// TwinCAT 3 PLC project PLC
// ProgramVersion: 3.1.4026.14
// CompilerDefines: VISU_USEPROPERTYINFO
// libraries:
//   Tc2_Standard, * (Beckhoff Automation GmbH)
//   Tc2_System, * (Beckhoff Automation GmbH)
//   Tc3_Analytics, * (Beckhoff Automation GmbH)
//   TcoCore, * (Vortex.Library)
//   TcoDrivesBeckhoff, * (Vortex.Library)
//   TcoElements, * (Vortex.Library)
//   TcoIo, * (Vortex.Library)
//   TcoPneumatics, * (Vortex.Library)
//   TcoUtilities, * (Vortex.Library)
//   VisuDialogs, * (System)
// project tree:
//   Components/ ST_MachineSetting.TcDUT (not stored)
//   Components/TcaCarrier/Structures/ TcaCarrierService.TcDUT (not stored), TcaCarrierConfig.TcDUT (not stored), TcaCarrierStatus.TcDUT
//   Components/TcaCarrier/Enumerations/ eTcaCarrierCmd.TcDUT (not stored), eTcaCarrierConfig.TcDUT (not stored)
//   Components/TcaCarrier/ ITcaCarrier.TcIO (not stored), TcaCarrier.TcPOU
//   Components/TcaCarrier/Tasks/ TcaCarrierModifyTask.TcPOU
//   Components/TcaPushButton/Enumerations/ eTcaPushButtonColor.TcDUT (not stored), eTcaPushButtonLightState.TcDUT (not stored)
//   Components/TcaPushButton/Structures/ TcaPushButtonStatus.TcDUT, TcaPushButtonRef.TcDUT, TcaPushButtonConfig.TcDUT, TcaPushButtonService.TcDUT (not stored)
//   Components/TcaPushButton/ TcaPushButton.TcPOU (not stored)
//   Components/TcaStorage/ E_ApproachDirection.TcDUT, eTcaStorageCmd.TcDUT (not stored), TcaRobotStorage.TcPOU (excluded from build), TcaStorage.TcPOU (not stored), TcaStorageRef.TcDUT (not stored)
//   Components/TcaTrolley/ CMD_Trolley.TcDUT (not stored), eTcaTrolleyCmd.TcDUT (not stored), TcaTrolley.TcPOU, TcaTrolleyRef.TcDUT
//   Components/TcaWorkpiecePlace/Enumerations/ eTcaWorkpiecePlaceProgress.TcDUT, eTcaWorkpiecePlaceStatus.TcDUT
//   Components/TcaWorkpiecePlace/Structures/ TcaWorkpiecePlaceService.TcDUT (not stored), TcaWorkpiecePlaceConfig.TcDUT, TcaWorkpiecePlaceStatus.TcDUT
//   Components/TcaWorkpiecePlace/ TcaWorkpiecePlace.TcPOU (not stored)
//   Components_RMTH/TcaEngelCasting/ Schnittstellenprotokoll.TcDUT (not stored), TcaEngelCastingCarrierInput.TcDUT (not stored), TcaEngelCastingCarrierJob.TcDUT (not stored), TcaEngelCastingCarrierJobStatus.TcDUT (not stored), TcaEngelCastingCarrierOutput.TcDUT (not stored), TcalEngelCastingCarrierStatus.TcDUT (not stored)
//   Components_RMTH/TcaLaserDistanceSenor/Structures/ TcaLaserDistanceSenorConfig.TcDUT, TcaLaserDistanceSenorRef.TcDUT (not stored), TcaLaserDistanceSenorStatus.TcDUT, TcaLaserDistanceSensorDataArrayEntry.TcDUT (not stored), TcaLaserDistanceSenorService.TcDUT
//   Components_RMTH/TcaLaserDistanceSenor/ TcaLaserDistanceSenor.TcPOU
//   Components_RMTH/TcaRackFeeder/Structures/ TcaRackFeederConfig.TcDUT, TcaRackFeederRef.TcDUT, TcaRackFeederService.TcDUT (not stored), TcaRackFeederStatus.TcDUT (not stored)
//   Components_RMTH/TcaRackFeeder/ TcaRackFeeder.TcPOU
//   Components_RMTH/TcaSafetyGate/ ISafetyComponent.TcIO (not stored), TcaSafetyGate.TcPOU (not stored)
//   Components_RMTH/TcaSafetyGate/Structures/ TcaSafetyGateConfig.TcDUT, TcaSafetyGateRef.TcDUT (not stored), TcaSafetyGateService.TcDUT (not stored), TcaSafetyGateStatus.TcDUT (not stored)
//   Components_RMTH/TcaSegmentDoor/Structures/ TcaSegmentDoorConfig.TcDUT, TcaSegmentDoorRef.TcDUT (not stored), TcaSegmentDoorService.TcDUT (not stored), TcaSegmentDoorStatus.TcDUT
//   Components_RMTH/TcaSegmentDoor/ TcaSegmentDoor.TcPOU (not stored)
//   Components_RMTH/TcaTwinSAFE/Structures/ TcaTwinSAFEConfig.TcDUT (not stored), TcaTwinSAFERef.TcDUT (not stored), TcaTwinSAFEService.TcDUT (not stored), TcaTwinSAFEStatus.TcDUT (not stored)
//   Components_RMTH/TcaTwinSAFE/ TcaTwinSAFE.TcPOU
//   / GlobalTextList.TcGTLO (not stored), PlcTask.TcTTO (not stored), Visualization Manager.TcVMO (not stored)
//   Items/ COLOR.TcDUT (not stored), E_Coordinate.TcDUT, ST_ComboboxEntry.TcDUT (not stored), ST_Coordinate.TcDUT, ST_WorkpieceType.TcDUT (not stored)
//   Program/Handling/Dialogs/ Handling_TeachRack_DlgContent.TcPOU (not stored)
//   Program/Handling/Sequences/ Handling_Teach.TcPOU, Handling_TeachRack.TcPOU, Handling_GroundMode.TcPOU (not stored), Handling_OpenDoor.TcPOU (not stored)
//   Program/ MAIN.TcPOU, Peripherie.TcPOU (not stored)
//   Program/Handling/ Handling.TcPOU (not stored), Handling_Components.TcPOU, Handling_Positions.TcPOU (not stored)
//   Template/Component_Cylinder/Base/ CylinderBase.TcPOU (not stored), TcoCylinderBase.TcPOU, TcoDoubleCylinderBase.TcPOU (not stored)
//   Template/Component_Cylinder/ ITcoCylinder.TcIO, TcoCylinder.TcPOU (not stored), TcoDoubleCylinder.TcPOU (not stored)
//   Template/Component_Cylinder/Structs/ CylinderConfig.TcDUT (not stored), CylinderStatus.TcDUT, TcoCylinderConfig.TcDUT (not stored), TcoCylinderStatus.TcDUT (not stored)
//   Template/Component_Cylinder/Tasks/ CylinderMoveTask.TcPOU (not stored), TcoCylinderMoveTask.TcPOU
//   Template/RackFeeder/ CMD_RackFeeder.TcDUT (not stored), E_RackFeederCmd.TcDUT, FB_RackFeeder.TcPOU (not stored)
//   Template/RackFeeder/Structure/ ST_RackFeederIO.TcDUT (not stored), ST_RackFeederJob.TcDUT (not stored), ST_StorageDock.TcDUT, ST_TrolleyDock.TcDUT
//   Template/Station/Data/ ST001_ProcessData.TcDUT, ST001_ProcessDataManager.TcPOU
//   Template/Station/ ST001.TcPOU (not stored), ST001_AutomatSequence.TcPOU, ST001_Components.TcDUT, ST001_ComponentsHandler.TcPOU (not stored), ST001_GroundSequence.TcPOU (not stored)
//   Template/Component_Carousell/Base/ TcoCarouselBase.TcPOU
//   Template/Component_Carousell/Structs/ eTcoCarouselDirection.TcDUT (not stored), TcoCarouselConfig.TcDUT (not stored), TcoCarouselStatus.TcDUT (not stored)
//   Template/Component_Carousell/Tasks/ TcoTurnTableTask.TcPOU (not stored)
//   Template/Component_Carousell/ TcoCarousel.TcPOU
//   Utilities/Component/Enumerations/ E_ComponentState.TcDUT (not stored), E_SafeState.TcDUT
//   Utilities/Component/ FB_Component.TcPOU (not stored), FB_ComponentPool.TcPOU
//   Utilities/Component/Interfaces/ ITF_Component.TcIO
//   Utilities/Component/Structures/ ST_ComponentVisu.TcDUT (not stored)
//   Utilities/Component/Visualisation/ Uc_Component.TcVIS
//   Utilities/EventLog/Base/ FB_LoggingProviderBase.TcPOU
//   Utilities/EventLog/Enumerations/ E_BoolFilter.TcDUT, E_FilterActive.TcDUT, E_LoggingProvider.TcDUT (not stored), E_LogLevel.TcDUT, E_Priority.TcDUT (not stored), ST_LoggingConfig.TcDUT
//   Utilities/EventLog/ E_Event.TcDUT (not stored), FB_EventLog.TcPOU (not stored)
//   Utilities/EventLog/Interface/ ITFLoggingProvider.TcIO (not stored), ITF_EventLog.TcIO
//   Utilities/EventLog/Structures/ ST_Event.TcDUT, ST_EventBase.TcDUT (not stored), ST_EventOutput.TcDUT, ST_EventVisu.TcDUT (not stored), ST_Log.TcDUT
//   Utilities/EventLog/Visualization/ Uc_EventLog.TcVIS, Uc_EventLogControl.TcDUT, Uc_EventLogControl.TcVIS, Uc_EventLogEntry.TcVIS, Uc_EventLogTable.TcDUT, Uc_EventLogTable.TcVIS
//   Utilities/Helpers/Color/ F_DWORD2CMYK.TcPOU, F_DWORD2RGB.TcPOU (not stored), F_RGB2CMYK.TcPOU (not stored), F_RGB2DWORD.TcPOU, F_TextColor.TcPOU (not stored), ST_Color.TcDUT, ST_ColorCMYK.TcDUT (not stored)
//   Utilities/Helpers/Concat/ Concat10.TcPOU, Concat2.TcPOU (not stored), Concat3.TcPOU, Concat4.TcPOU, Concat5.TcPOU, Concat6.TcPOU, Concat7.TcPOU (not stored), Concat8.TcPOU, Concat9.TcPOU, ConcatArray.TcPOU
//   Utilities/Helpers/ E_OperationResult.TcDUT (not stored), FB_GetTimeString.TcPOU (excluded from build), FB_Pulse.TcPOU, FB_TON_RMTH.TcPOU, F_BYTE_TO_INT.TcPOU, F_BYTE_TO_REAL.TcPOU (not stored), F_DT_TO_STRING.TcPOU (not stored), F_GetAdsPort.TcPOU (not stored), F_GetPlcCycleTime.TcPOU, F_GetSystemTime64.TcPOU, F_TO_STRING.TcPOU, P_FilePath.TcPOU (not stored), P_System.TcPOU, ST_DefaultPulse.TcDUT (not stored), ST_PlcSystemInfo.TcDUT (not stored)
//   Utilities/ HexColor.TcGVL, Statics.TcGVL, StaticsConstant.TcGVL (not stored)
//   Utilities/List/ FB_List.TcPOU (not stored)
//   Utilities/List/Structures/ ST_Listentry.TcDUT (not stored), Uc_List.TcDUT
//   Utilities/List/Visu/ Uc_EntryDetail.TcVIS (not stored), Uc_List.TcVIS, Uc_Listentry.TcVIS
//   Utilities/Sequencer/Enumeration/ E_SequenceState.TcDUT
//   Utilities/Sequencer/ FB_Sequence.TcPOU
// real-time tasks:
//   TASK PlcTask: cycle T#10ms, priority 20, ADS port 350
// motion (NC):
//   TASK NC-Task 1 SAF: cycle T#2ms, priority 4, ADS port 501
//   TASK NC-Task 1 SVB: cycle T#10ms, priority 8, ADS port 511
//   AXIS Oven B CH1 (id 14)
//     Dynamic: Acceleration=282800000, Deceleration=282800000, Jerk=2.85628e+17
//     Velo: RefSearch=25, RefSync=25, SlowManual=14, FastManual=28, Maximum=28
//     PositionAreaControl: Enable=false
//     TargetPosControl: Enable=false
//     OtherSettings: AllowMotionCmdToSlave=true
//     encoder EncType=7
//       EncPara: ScaleFactorNumerator=0.001879, Offset=-1.4, MaxCount=#x0000ffff, ReferenceSystem=1
//     drive DrvType=23
//       Analog: VeloReferenz=28, TorqueSetpointScale=10, ScaleFactorActTorque=0.1
//       TimeComp: TaskDelayCycles=1
//     controller CtrType=1
//       CtrPara: PriorControlFactor=1
//         PosDiffControl: Enable=false
//         Observer: BandWidth=20
//   AXIS Oven B CH2 (id 15)
//     Dynamic: Acceleration=282800000, Deceleration=282800000, Jerk=2.85628e+17
//     Velo: RefSearch=25, RefSync=25, SlowManual=14, FastManual=28, Maximum=28
//     PositionAreaControl: Enable=false
//     TargetPosControl: Enable=false
//     OtherSettings: AllowMotionCmdToSlave=true
//     encoder EncType=7
//       EncPara: ScaleFactorNumerator=0.001879, Offset=-1.4, MaxCount=#x0000ffff, ReferenceSystem=1
//     drive DrvType=23
//       Analog: VeloReferenz=28, TorqueSetpointScale=10, ScaleFactorActTorque=0.1
//       TimeComp: TaskDelayCycles=1
//     controller CtrType=1
//       CtrPara: PriorControlFactor=1
//         PosDiffControl: Enable=false
//         Observer: BandWidth=20
//   AXIS Rackfeeder X (id 16)
//     Dynamic: Acceleration=2461.9275, Deceleration=2461.9275, Jerk=7385.7825
//     Velo: RefSearch=16.41285, RefSync=16.41285, SlowManual=10, FastManual=60, Fast=1641.285, Maximum=1641.285
//     OtherSettings: AllowMotionCmdToSlave=true
//     encoder EncType=8
//       EncPara: ScaleFactorNumerator=150, ScaleFactorDenominator=10485760, MaxCount=#xffffffff
//     drive DrvType=9
//       DrvPara: MaxCount=#xffffffff, DriveControlDWord=#x00030100
//         Analog: VeloReferenz=1805.4135, VeloScale=1.02400649589962, TorqueSetpointScale=10, ScaleFactorActTorque=0.1
//         TimeComp: TaskDelayCycles=1
//     controller CtrType=1
//       CtrPara: PriorControlFactor=1
//         Observer: BandWidth=20
//   AXIS Rackfeeder Y (id 17)
//     Dynamic: Acceleration=2256.7665, Deceleration=2256.7665, Jerk=6770.2995
//     Velo: RefSearch=15.04511, RefSync=15.04511, SlowManual=10, FastManual=60, Fast=1504.511, Maximum=1504.511
//     OtherSettings: AllowMotionCmdToSlave=true
//     encoder EncType=8
//       EncPara: ScaleFactorNumerator=220, ScaleFactorDenominator=16777216, MaxCount=#xffffffff
//     drive DrvType=9
//       DrvPara: MaxCount=#xffffffff, DriveControlDWord=#x00030100
//         Analog: VeloReferenz=1654.9621, VeloScale=1.02400649589962, TorqueSetpointScale=10, ScaleFactorActTorque=0.1
//         TimeComp: TaskDelayCycles=1
//     controller CtrType=1
//       CtrPara: PriorControlFactor=1
//         Observer: BandWidth=20
//   AXIS Rackfeeder Teleskop (id 18)
//     OtherSettings: AllowMotionCmdToSlave=true
//     encoder EncType=8
//       EncPara: MaxCount=#xffffffff
//     drive DrvType=9
//       DrvPara: MaxCount=#xffffffff, DriveControlDWord=#x00030100
//         Analog: VeloScale=1.02400649589962, TorqueSetpointScale=10, ScaleFactorActTorque=0.1
//         TimeComp: TaskDelayCycles=1
//     controller CtrType=1
//       CtrPara: PriorControlFactor=1
//         Observer: BandWidth=20
//   AXIS Oven B (id 21)
//     Dynamic: Acceleration=1231.0125, Deceleration=1231.0125, Jerk=3693.0375
//     Velo: RefSearch=8.20675, RefSync=8.20675, SlowManual=20, FastManual=120, Fast=820.675, Maximum=820.675
//     OtherSettings: AllowMotionCmdToSlave=true
//     encoder EncType=8
//       EncPara: ScaleFactorNumerator=120, ScaleFactorDenominator=16777216, Inverse=true, MaxCount=#xffffffff
//     drive DrvType=9
//       DrvPara: Inverse=true, MaxCount=#xffffffff, DriveControlDWord=#x00030100
//         Analog: VeloReferenz=902.7425, VeloScale=1.02400649589962, TorqueSetpointScale=10, ScaleFactorActTorque=0.1
//         TimeComp: TaskDelayCycles=1
//     controller CtrType=1
//       CtrPara: PriorControlFactor=1
//         Observer: BandWidth=20
//   AXIS Oven A (id 20)
//     Dynamic: Acceleration=1231.0125, Deceleration=1231.0125, Jerk=3693.0375
//     Velo: RefSearch=8.20675, RefSync=8.20675, SlowManual=20, FastManual=120, Fast=820.675, Maximum=820.675
//     OtherSettings: AllowMotionCmdToSlave=true
//     encoder EncType=8
//       EncPara: ScaleFactorNumerator=120, ScaleFactorDenominator=16777216, Inverse=true, MaxCount=#xffffffff
//     drive DrvType=9
//       DrvPara: Inverse=true, MaxCount=#xffffffff, DriveControlDWord=#x00030100
//         Analog: VeloReferenz=902.7425, VeloScale=1.02400649589962, TorqueSetpointScale=10, ScaleFactorActTorque=0.1
//         TimeComp: TaskDelayCycles=1
//     controller CtrType=1
//       CtrPara: PriorControlFactor=1
//         Observer: BandWidth=20
//   AXIS Oven A CH1 (id 1)
//     Dynamic: Acceleration=282800000, Deceleration=282800000, Jerk=2.85628e+17, DelayTime=0.01, OverrideType=4
//     Velo: RefSearch=25, RefSync=25, SlowManual=14, FastManual=28, Maximum=28
//     PositionAreaControl: Enable=false
//     TargetPosControl: Enable=false
//     OtherSettings: AllowMotionCmdToSlave=true
//     encoder EncType=7
//       EncPara: ScaleFactorNumerator=0.001879, Offset=-1.4, EncMode=1, MaxCount=#x0000ffff, ReferenceSystem=1
//         FilterTime: TVelo=0.1
//         SoftEndMinControl: Range=-5
//         SoftEndMaxControl: Range=30
//         ActPosCorrection: Enable=true, Time=1
//     drive DrvType=23
//       Analog: VeloReferenz=28, TorqueSetpointScale=10, ScaleFactorActTorque=0.1
//       TimeComp: TaskDelayCycles=1
//     controller CtrType=1
//       CtrPara: PriorControlFactor=1
//         PosDiffControl: Enable=false
//         Observer: BandWidth=20
//   AXIS Oven A CH2 (id 13)
//     Dynamic: Acceleration=282800000, Deceleration=282800000, Jerk=2.85628e+17
//     Velo: RefSearch=25, RefSync=25, SlowManual=14, FastManual=28, Maximum=28
//     PositionAreaControl: Enable=false
//     TargetPosControl: Enable=false
//     OtherSettings: AllowMotionCmdToSlave=true
//     encoder EncType=7
//       EncPara: ScaleFactorNumerator=0.001879, Offset=-1.4, MaxCount=#x0000ffff, ReferenceSystem=1
//     drive DrvType=23
//       Analog: VeloReferenz=28, TorqueSetpointScale=10, ScaleFactorActTorque=0.1
//       TimeComp: TaskDelayCycles=1
//     controller CtrType=1
//       CtrPara: PriorControlFactor=1
//         PosDiffControl: Enable=false
//         Observer: BandWidth=20
// I/O:
//   DEVICE Gerät 3 (EtherCAT), AmsNetId 5.24.124.74.4.1
//     Klemme 1 (EK1100) [EK1100 EtherCAT-Koppler (2A E-Bus)]
//       Klemme 33 (EL6910) [EL6910, TwinSAFE PLC]
//       Klemme 3 (EL1904) [EL1904, 4 K. Safety Eingang 24V, TwinSAFE]
//         modules: Module 1 (FSOES)
//       Klemme 4 (EL2904) [EL2904, 4 K. Safety Ausgang 24V, 0.5A, TwinSAFE]
//         modules: Module 1 (FSOES), Module 2 (DO)
//       Klemme 5 (EL1104) [EL1104 4K. Dig. Eingang 24V, 3ms, Sensorversorgung]
//       Klemme 6 (EL1104) [EL1104 4K. Dig. Eingang 24V, 3ms, Sensorversorgung]
//       Klemme 7 (EL6224) [EL6224 (IO Link Master)]
//       ENGEL Interface (EL1008) [EL1008 8K. Dig. Eingang 24V, 3ms]
//       ENGEL Interface (EL2624) [EL2624 4K. Relais Ausgang, Schließer (125V AC / 30V DC)]
//       Ovens (EK1122) [EK1122 2-Port EtherCAT-Abzweig]
//         Oven_A (EK1100) [EK1100 EtherCAT-Koppler (2A E-Bus)]
//           Klemme 10 (EL1904) [EL1904, 4 K. Safety Eingang 24V, TwinSAFE]
//             modules: Module 1 (FSOES)
//           Klemme 11 (EL2904) [EL2904, 4 K. Safety Ausgang 24V, 0.5A, TwinSAFE]
//             modules: Module 1 (FSOES), Module 2 (DO)
//           Klemme 12 (EL7332) [EL7332 2K. DC-Motor-Endstufe (24V, 1.5A)]
//           Klemme 13 (EL3062-0030) [EL3062-0030 2K.Ana. Eingang 0-30V]
//           Klemme 14 (EL1004) [EL1004 4K. Dig. Eingang 24V, 3ms]
//           Klemme 15 (EL2004) [EL2004 4K. Dig. Ausgang 24V, 0.5A]
//           Klemme 16 (EL9010) [EL9010 Endklemme]
//         Oven_B (EK1100) [EK1100 EtherCAT-Koppler (2A E-Bus)]
//           Klemme 18 (EL1904) [EL1904, 4 K. Safety Eingang 24V, TwinSAFE]
//             modules: Module 1 (FSOES)
//           Klemme 19 (EL2904) [EL2904, 4 K. Safety Ausgang 24V, 0.5A, TwinSAFE]
//             modules: Module 1 (FSOES), Module 2 (DO)
//           Klemme 20 (EL7332) [EL7332 2K. DC-Motor-Endstufe (24V, 1.5A)]
//           Klemme 21 (EL3062-0030) [EL3062-0030 2K.Ana. Eingang 0-30V]
//           Klemme 22 (EL1004) [EL1004 4K. Dig. Eingang 24V, 3ms]
//           Klemme 23 (EL2004) [EL2004 4K. Dig. Ausgang 24V, 0.5A]
//           Klemme 61 (EL9010) [EL9010 Endklemme]
//       Storage|Casting (EK1122) [EK1122 2-Port EtherCAT-Abzweig]
//         Storage (EK1100)
//     RackFeeder_X_Y (AX5206-0000-0215) [AX5206-0000-0215 EtherCAT Drive (SoE, 2 Ch.)]
//       Klemme 27 (AX5805) [AX5805 (Safety Drive Option)]
//         modules: Module 1 (Safety Process Data, 2 axis), Module 2 (Standard Process Data, 2 axis)
//     Rackfeeder_Teleskop (AX5203-0000-0215) [AX5203-0000-0215 EtherCAT Drive (SoE, 2 Ch.)]
//       Klemme 29 (AX5805) [AX5805 (Safety Drive Option)]
//         modules: Module 1 (Safety Process Data, 2 axis), Module 2 (Standard Process Data, 2 axis)
//     OvenDoor_A_B (AX5206-0000-0215) [AX5206-0000-0215 EtherCAT Drive (SoE, 2 Ch.)]
//       Klemme 31 (AX5805) [AX5805 (Safety Drive Option)]
//         modules: Module 1 (Safety Process Data, 2 axis), Module 2 (Standard Process Data, 2 axis)
// variable links:
//   Device 3 (EtherCAT) <-> Device 3 (EtherCAT)/OvenDoor_A_B (AX5206-0000-0215)/Term 31 (AX5805)
//     Term 1 (EK1100)/Term 33 (EL6910)/ConnectionInputs/TwinSafeMain.Oven (AX5805) - Module 1 (Safety Process Data, 2 axis)_120 TxPDO <-> Module 1 (Safety Process Data, 2 axis)/Outputs (Controlword)/FSOE
//     Term 1 (EK1100)/Term 33 (EL6910)/ConnectionOutputs/TwinSafeMain.Oven (AX5805) - Module 1 (Safety Process Data, 2 axis)_120 RxPDO <-> Module 1 (Safety Process Data, 2 axis)/Inputs (Statusword)/FSOE
//   Device 3 (EtherCAT) <-> Device 3 (EtherCAT)/RackFeeder_X_Y (AX5206-0000-0215)/Term 27 (AX5805)
//     Term 1 (EK1100)/Term 33 (EL6910)/ConnectionInputs/TwinSafeMain.Rackfeeder_XY (AX5805) - Module 1 (Safety Process Data, 2 axis)_118 TxPDO <-> Module 1 (Safety Process Data, 2 axis)/Outputs (Controlword)/FSOE
//     Term 1 (EK1100)/Term 33 (EL6910)/ConnectionOutputs/TwinSafeMain.Rackfeeder_XY (AX5805) - Module 1 (Safety Process Data, 2 axis)_118 RxPDO <-> Module 1 (Safety Process Data, 2 axis)/Inputs (Statusword)/FSOE
//   Device 3 (EtherCAT) <-> Device 3 (EtherCAT)/Rackfeeder_Teleskop (AX5203-0000-0215)/Term 29 (AX5805)
//     Term 1 (EK1100)/Term 33 (EL6910)/ConnectionInputs/TwinSafeMain.Rackfeeder_Tele (AX5805) - Module 1 (Safety Process Data, 2 axis)_119 TxPDO <-> Module 1 (Safety Process Data, 2 axis)/Outputs (Controlword)/FSOE
//     Term 1 (EK1100)/Term 33 (EL6910)/ConnectionOutputs/TwinSafeMain.Rackfeeder_Tele (AX5805) - Module 1 (Safety Process Data, 2 axis)_119 RxPDO <-> Module 1 (Safety Process Data, 2 axis)/Inputs (Statusword)/FSOE
//   Device 3 (EtherCAT) <-> Device 3 (EtherCAT)/Term 1 (EK1100)/Ovens (EK1122)/Oven_A (EK1100)/Term 10 (EL1904)
//     Term 1 (EK1100)/Term 33 (EL6910)/ConnectionInputs/TwinSafeMain.Oven A (EL1904) - Module 1 (FSOES)_14 TxPDO <-> Module 1 (FSOES)/RxPDO/FSOE
//     Term 1 (EK1100)/Term 33 (EL6910)/ConnectionOutputs/TwinSafeMain.Oven A (EL1904) - Module 1 (FSOES)_14 RxPDO <-> Module 1 (FSOES)/TxPDO/FSOE
//   Device 3 (EtherCAT) <-> Device 3 (EtherCAT)/Term 1 (EK1100)/Ovens (EK1122)/Oven_A (EK1100)/Term 11 (EL2904)
//     Term 1 (EK1100)/Term 33 (EL6910)/ConnectionInputs/TwinSafeMain.Oven A (EL2904) - Module 1 (FSOES)_111 TxPDO <-> Module 1 (FSOES)/RxPDO/FSOE
//     Term 1 (EK1100)/Term 33 (EL6910)/ConnectionOutputs/TwinSafeMain.Oven A (EL2904) - Module 1 (FSOES)_111 RxPDO <-> Module 1 (FSOES)/TxPDO/FSOE
//   Device 3 (EtherCAT) <-> Device 3 (EtherCAT)/Term 1 (EK1100)/Ovens (EK1122)/Oven_B (EK1100)/Term 18 (EL1904)
//     Term 1 (EK1100)/Term 33 (EL6910)/ConnectionOutputs/TwinSafeMain.Oven B (EL1904) - Module 1 (FSOES)_16 RxPDO <-> Module 1 (FSOES)/TxPDO/FSOE
//   Device 3 (EtherCAT) <-> Device 3 (EtherCAT)/Term 1 (EK1100)/Ovens (EK1122)/Oven_B (EK1100)/Term 19 (EL2904)
//     Term 1 (EK1100)/Term 33 (EL6910)/ConnectionInputs/TwinSafeMain.Oven B (EL2904) - Module 1 (FSOES)_112 TxPDO <-> Module 1 (FSOES)/RxPDO/FSOE
//     Term 1 (EK1100)/Term 33 (EL6910)/ConnectionOutputs/TwinSafeMain.Oven B (EL2904) - Module 1 (FSOES)_112 RxPDO <-> Module 1 (FSOES)/TxPDO/FSOE
//   Device 3 (EtherCAT) <-> Device 3 (EtherCAT)/Term 1 (EK1100)/Term 3 (EL1904)
//     Term 1 (EK1100)/Term 33 (EL6910)/ConnectionInputs/TwinSafeMain.MAIN (EL1904) - Module 1 (FSOES)_12 TxPDO <-> Module 1 (FSOES)/RxPDO/FSOE
//     Term 1 (EK1100)/Term 33 (EL6910)/ConnectionOutputs/TwinSafeMain.MAIN (EL1904) - Module 1 (FSOES)_12 RxPDO <-> Module 1 (FSOES)/TxPDO/FSOE
//   Device 3 (EtherCAT) <-> Device 3 (EtherCAT)/Term 1 (EK1100)/Term 33 (EL6910)
//     Term 1 (EK1100)/Ovens (EK1122)/Oven_B (EK1100)/Term 18 (EL1904)/Module 1 (FSOES)/RxPDO/FSOE <-> ConnectionInputs/TwinSafeMain.Oven B (EL1904) - Module 1 (FSOES)_16 TxPDO
//   Device 3 (EtherCAT) <-> Device 3 (EtherCAT)/Term 1 (EK1100)/Term 4 (EL2904)
//     Term 1 (EK1100)/Term 33 (EL6910)/ConnectionInputs/TwinSafeMain.MAIN (EL2904) - Module 1 (FSOES)_13 TxPDO <-> Module 1 (FSOES)/RxPDO/FSOE
//     Term 1 (EK1100)/Term 33 (EL6910)/ConnectionOutputs/TwinSafeMain.MAIN (EL2904) - Module 1 (FSOES)_13 RxPDO <-> Module 1 (FSOES)/TxPDO/FSOE
//   NC-Task 1 SAF/Axes/Oven A <-> Device 3 (EtherCAT)/OvenDoor_A_B (AX5206-0000-0215)
//     Drive/Inputs/In/nDataIn1 <-> AT 1/Following distance
//     Drive/Inputs/In/nDcOutputTime <-> InfoData/DcOutputShift
//     Drive/Inputs/In/nState1 <-> AT 1/Drive status word @bit 8
//     Drive/Inputs/In/nState2 <-> AT 1/Drive status word
//     Drive/Inputs/In/nState4 @bit 1 <-> WcState/InputToggle
//     Drive/Inputs/In/nState4 <-> WcState/WcState
//     Drive/Outputs/Out/nCtrl1 <-> MDT 1/Master control word @bit 8
//     Drive/Outputs/Out/nDataOut1 <-> MDT 1/Position command value
//     Enc/Inputs/In/nDataIn1 <-> AT 1/Position feedback 1 value
//     Enc/Inputs/In/nDcInputTime <-> InfoData/DcInputShift
//     Enc/Inputs/In/nState4 @bit 1 <-> WcState/InputToggle
//     Enc/Inputs/In/nState4 <-> WcState/WcState
//   NC-Task 1 SAF/Axes/Oven A CH1 <-> Device 3 (EtherCAT)/Term 1 (EK1100)/Ovens (EK1122)/Oven_A (EK1100)/Term 12 (EL7332)
//     Drive/Inputs/In/nState1 @bit 3 <-> DCM Status Channel 1/Status/Error
//     Drive/Inputs/In/nState1 @bit 5 <-> DCM Status Channel 1/Status/Moving negative
//     Drive/Inputs/In/nState1 @bit 4 <-> DCM Status Channel 1/Status/Moving positive
//     Drive/Inputs/In/nState1 @bit 1 <-> DCM Status Channel 1/Status/Ready
//     Drive/Inputs/In/nState1 <-> DCM Status Channel 1/Status/Ready to enable
//     Drive/Inputs/In/nState1 @bit 6 <-> DCM Status Channel 1/Status/Torque reduced
//     Drive/Inputs/In/nState1 @bit 2 <-> DCM Status Channel 1/Status/Warning
//     Drive/Inputs/In/nState2 @bit 3 <-> DCM Status Channel 1/Status/Digital input 1
//     Drive/Inputs/In/nState2 @bit 4 <-> DCM Status Channel 1/Status/Digital input 2
//     Drive/Inputs/In/nState2 @bit 5 <-> DCM Status Channel 1/Status/Sync error
//     Drive/Inputs/In/nState2 @bit 7 <-> DCM Status Channel 1/Status/TxPDO Toggle
//     Drive/Inputs/In/nState4 @bit 1 <-> WcState/InputToggle
//     Drive/Inputs/In/nState4 <-> WcState/WcState
//     Drive/Outputs/Out/nCtrl1 <-> DCM Control Channel 1/Control/Enable
//     Drive/Outputs/Out/nCtrl1 @bit 2 <-> DCM Control Channel 1/Control/Reduce torque
//     Drive/Outputs/Out/nCtrl1 @bit 1 <-> DCM Control Channel 1/Control/Reset
//     Drive/Outputs/Out/nDataOut2[0] <-> DCM Velocity Channel 1/Velocity
//   NC-Task 1 SAF/Axes/Oven A CH1 <-> Device 3 (EtherCAT)/Term 1 (EK1100)/Ovens (EK1122)/Oven_A (EK1100)/Term 13 (EL3062-0030)
//     Enc/Inputs/In/nDataIn1[0] <-> AI Standard Channel 1/Value
//     Enc/Inputs/In/nState4 @bit 1 <-> WcState/InputToggle
//     Enc/Inputs/In/nState4 <-> WcState/WcState
//   NC-Task 1 SAF/Axes/Oven A CH2 <-> Device 3 (EtherCAT)/Term 1 (EK1100)/Ovens (EK1122)/Oven_A (EK1100)/Term 12 (EL7332)
//     Drive/Inputs/In/nState1 @bit 3 <-> DCM Status Channel 2/Status/Error
//     Drive/Inputs/In/nState1 @bit 5 <-> DCM Status Channel 2/Status/Moving negative
//     Drive/Inputs/In/nState1 @bit 4 <-> DCM Status Channel 2/Status/Moving positive
//     Drive/Inputs/In/nState1 @bit 1 <-> DCM Status Channel 2/Status/Ready
//     Drive/Inputs/In/nState1 <-> DCM Status Channel 2/Status/Ready to enable
//     Drive/Inputs/In/nState1 @bit 6 <-> DCM Status Channel 2/Status/Torque reduced
//     Drive/Inputs/In/nState1 @bit 2 <-> DCM Status Channel 2/Status/Warning
//     Drive/Inputs/In/nState2 @bit 3 <-> DCM Status Channel 2/Status/Digital input 1
//     Drive/Inputs/In/nState2 @bit 4 <-> DCM Status Channel 2/Status/Digital input 2
//     Drive/Inputs/In/nState2 @bit 5 <-> DCM Status Channel 2/Status/Sync error
//     Drive/Inputs/In/nState2 @bit 7 <-> DCM Status Channel 2/Status/TxPDO Toggle
//     Drive/Inputs/In/nState4 @bit 1 <-> WcState/InputToggle
//     Drive/Inputs/In/nState4 <-> WcState/WcState
//     Drive/Outputs/Out/nCtrl1 <-> DCM Control Channel 2/Control/Enable
//     Drive/Outputs/Out/nCtrl1 @bit 2 <-> DCM Control Channel 2/Control/Reduce torque
//     Drive/Outputs/Out/nCtrl1 @bit 1 <-> DCM Control Channel 2/Control/Reset
//     Drive/Outputs/Out/nDataOut2[0] <-> DCM Velocity Channel 2/Velocity
//   NC-Task 1 SAF/Axes/Oven A CH2 <-> Device 3 (EtherCAT)/Term 1 (EK1100)/Ovens (EK1122)/Oven_A (EK1100)/Term 13 (EL3062-0030)
//     Enc/Inputs/In/nDataIn1[0] <-> AI Standard Channel 2/Value
//     Enc/Inputs/In/nState4 @bit 1 <-> WcState/InputToggle
//     Enc/Inputs/In/nState4 <-> WcState/WcState
//   NC-Task 1 SAF/Axes/Oven B <-> Device 3 (EtherCAT)/OvenDoor_A_B (AX5206-0000-0215)
//     Drive/Inputs/In/nDataIn1 <-> AT 2/Following distance
//     Drive/Inputs/In/nDcOutputTime <-> InfoData/DcOutputShift
//     Drive/Inputs/In/nState1 <-> AT 2/Drive status word @bit 8
//     Drive/Inputs/In/nState2 <-> AT 2/Drive status word
//     Drive/Inputs/In/nState4 @bit 1 <-> WcState/InputToggle
//     Drive/Inputs/In/nState4 <-> WcState/WcState
//     Drive/Outputs/Out/nCtrl1 <-> MDT 2/Master control word @bit 8
//     Drive/Outputs/Out/nDataOut1 <-> MDT 2/Position command value
//     Enc/Inputs/In/nDataIn1 <-> AT 2/Position feedback 1 value
//     Enc/Inputs/In/nDcInputTime <-> InfoData/DcInputShift
//     Enc/Inputs/In/nState4 @bit 1 <-> WcState/InputToggle
//     Enc/Inputs/In/nState4 <-> WcState/WcState
//   NC-Task 1 SAF/Axes/Oven B CH1 <-> Device 3 (EtherCAT)/Term 1 (EK1100)/Ovens (EK1122)/Oven_B (EK1100)/Term 20 (EL7332)
//     Drive/Inputs/In/nState1 @bit 3 <-> DCM Status Channel 1/Status/Error
//     Drive/Inputs/In/nState1 @bit 5 <-> DCM Status Channel 1/Status/Moving negative
//     Drive/Inputs/In/nState1 @bit 4 <-> DCM Status Channel 1/Status/Moving positive
//     Drive/Inputs/In/nState1 @bit 1 <-> DCM Status Channel 1/Status/Ready
//     Drive/Inputs/In/nState1 <-> DCM Status Channel 1/Status/Ready to enable
//     Drive/Inputs/In/nState1 @bit 6 <-> DCM Status Channel 1/Status/Torque reduced
//     Drive/Inputs/In/nState1 @bit 2 <-> DCM Status Channel 1/Status/Warning
//     Drive/Inputs/In/nState2 @bit 3 <-> DCM Status Channel 1/Status/Digital input 1
//     Drive/Inputs/In/nState2 @bit 4 <-> DCM Status Channel 1/Status/Digital input 2
//     Drive/Inputs/In/nState2 @bit 5 <-> DCM Status Channel 1/Status/Sync error
//     Drive/Inputs/In/nState2 @bit 7 <-> DCM Status Channel 1/Status/TxPDO Toggle
//     Drive/Inputs/In/nState4 @bit 1 <-> WcState/InputToggle
//     Drive/Inputs/In/nState4 <-> WcState/WcState
//     Drive/Outputs/Out/nCtrl1 <-> DCM Control Channel 1/Control/Enable
//     Drive/Outputs/Out/nCtrl1 @bit 2 <-> DCM Control Channel 1/Control/Reduce torque
//     Drive/Outputs/Out/nCtrl1 @bit 1 <-> DCM Control Channel 1/Control/Reset
//     Drive/Outputs/Out/nDataOut2[0] <-> DCM Velocity Channel 1/Velocity
//   NC-Task 1 SAF/Axes/Oven B CH1 <-> Device 3 (EtherCAT)/Term 1 (EK1100)/Ovens (EK1122)/Oven_B (EK1100)/Term 21 (EL3062-0030)
//     Enc/Inputs/In/nDataIn1[0] <-> AI Standard Channel 1/Value
//     Enc/Inputs/In/nState4 @bit 1 <-> WcState/InputToggle
//     Enc/Inputs/In/nState4 <-> WcState/WcState
//   NC-Task 1 SAF/Axes/Oven B CH2 <-> Device 3 (EtherCAT)/Term 1 (EK1100)/Ovens (EK1122)/Oven_B (EK1100)/Term 20 (EL7332)
//     Drive/Inputs/In/nState1 @bit 3 <-> DCM Status Channel 2/Status/Error
//     Drive/Inputs/In/nState1 @bit 5 <-> DCM Status Channel 2/Status/Moving negative
//     Drive/Inputs/In/nState1 @bit 4 <-> DCM Status Channel 2/Status/Moving positive
//     Drive/Inputs/In/nState1 @bit 1 <-> DCM Status Channel 2/Status/Ready
//     Drive/Inputs/In/nState1 <-> DCM Status Channel 2/Status/Ready to enable
//     Drive/Inputs/In/nState1 @bit 6 <-> DCM Status Channel 2/Status/Torque reduced
//     Drive/Inputs/In/nState1 @bit 2 <-> DCM Status Channel 2/Status/Warning
//     Drive/Inputs/In/nState2 @bit 3 <-> DCM Status Channel 2/Status/Digital input 1
//     Drive/Inputs/In/nState2 @bit 4 <-> DCM Status Channel 2/Status/Digital input 2
//     Drive/Inputs/In/nState2 @bit 5 <-> DCM Status Channel 2/Status/Sync error
//     Drive/Inputs/In/nState2 @bit 7 <-> DCM Status Channel 2/Status/TxPDO Toggle
//     Drive/Inputs/In/nState4 @bit 1 <-> WcState/InputToggle
//     Drive/Inputs/In/nState4 <-> WcState/WcState
//     Drive/Outputs/Out/nCtrl1 <-> DCM Control Channel 2/Control/Enable
//     Drive/Outputs/Out/nCtrl1 @bit 2 <-> DCM Control Channel 2/Control/Reduce torque
//     Drive/Outputs/Out/nCtrl1 @bit 1 <-> DCM Control Channel 2/Control/Reset
//     Drive/Outputs/Out/nDataOut2[0] <-> DCM Velocity Channel 2/Velocity
//   NC-Task 1 SAF/Axes/Oven B CH2 <-> Device 3 (EtherCAT)/Term 1 (EK1100)/Ovens (EK1122)/Oven_B (EK1100)/Term 21 (EL3062-0030)
//     Enc/Inputs/In/nDataIn1[0] <-> AI Standard Channel 2/Value
//     Enc/Inputs/In/nState4 @bit 1 <-> WcState/InputToggle
//     Enc/Inputs/In/nState4 <-> WcState/WcState
//   NC-Task 1 SAF/Axes/Rackfeeder Teleskop <-> Device 3 (EtherCAT)/Rackfeeder_Teleskop (AX5203-0000-0215)
//     Drive/Inputs/In/nDataIn1 <-> AT 1/Following distance
//     Drive/Inputs/In/nDcOutputTime <-> InfoData/DcOutputShift
//     Drive/Inputs/In/nState1 <-> AT 1/Drive status word @bit 8
//     Drive/Inputs/In/nState2 <-> AT 1/Drive status word
//     Drive/Inputs/In/nState4 @bit 1 <-> WcState/InputToggle
//     Drive/Inputs/In/nState4 <-> WcState/WcState
//     Drive/Outputs/Out/nCtrl1 <-> MDT 1/Master control word @bit 8
//     Drive/Outputs/Out/nDataOut1 <-> MDT 1/Position command value
//     Enc/Inputs/In/nDataIn1 <-> AT 1/Position feedback 1 value
//     Enc/Inputs/In/nDcInputTime <-> InfoData/DcInputShift
//     Enc/Inputs/In/nState4 @bit 1 <-> WcState/InputToggle
//     Enc/Inputs/In/nState4 <-> WcState/WcState
//   NC-Task 1 SAF/Axes/Rackfeeder X <-> Device 3 (EtherCAT)/RackFeeder_X_Y (AX5206-0000-0215)
//     Drive/Inputs/In/nDataIn1 <-> AT 1/Following distance
//     Drive/Inputs/In/nDcOutputTime <-> InfoData/DcOutputShift
//     Drive/Inputs/In/nState1 <-> AT 1/Drive status word @bit 8
//     Drive/Inputs/In/nState2 <-> AT 1/Drive status word
//     Drive/Inputs/In/nState4 @bit 1 <-> WcState/InputToggle
//     Drive/Inputs/In/nState4 <-> WcState/WcState
//     Drive/Outputs/Out/nCtrl1 <-> MDT 1/Master control word @bit 8
//     Drive/Outputs/Out/nDataOut1 <-> MDT 1/Position command value
//     Enc/Inputs/In/nDataIn1 <-> AT 1/Position feedback 1 value
//     Enc/Inputs/In/nDcInputTime <-> InfoData/DcInputShift
//     Enc/Inputs/In/nState4 @bit 1 <-> WcState/InputToggle
//     Enc/Inputs/In/nState4 <-> WcState/WcState
//   NC-Task 1 SAF/Axes/Rackfeeder Y <-> Device 3 (EtherCAT)/RackFeeder_X_Y (AX5206-0000-0215)
//     Drive/Inputs/In/nDataIn1 <-> AT 2/Following distance
//     Drive/Inputs/In/nDcOutputTime <-> InfoData/DcOutputShift
//     Drive/Inputs/In/nState1 <-> AT 2/Drive status word @bit 8
//     Drive/Inputs/In/nState2 <-> AT 2/Drive status word
//     Drive/Inputs/In/nState4 @bit 1 <-> WcState/InputToggle
//     Drive/Inputs/In/nState4 <-> WcState/WcState
//     Drive/Outputs/Out/nCtrl1 <-> MDT 2/Master control word @bit 8
//     Drive/Outputs/Out/nDataOut1 <-> MDT 2/Position command value
//     Enc/Inputs/In/nDataIn1 <-> AT 2/Position feedback 1 value
//     Enc/Inputs/In/nDcInputTime <-> InfoData/DcInputShift
//     Enc/Inputs/In/nState4 @bit 1 <-> WcState/InputToggle
//     Enc/Inputs/In/nState4 <-> WcState/WcState
//   PLC/PLC Instance <-> Device 3 (EtherCAT)/Term 1 (EK1100)/Ovens (EK1122)/Oven_A (EK1100)/Term 14 (EL1004)
//     PlcTask Inputs/MAIN._Peripherie._Handling._components.SafetyGateRef_A.LockButton.Button <-> Channel 3/MAIN._Peripherie._Handling._components.SafetyGateRef_A.LockButton.Button
//     PlcTask Inputs/MAIN._Peripherie._Handling._components.SafetyGateRef_A.RequestButton.Button <-> Channel 2/MAIN._Peripherie._Handling._components.SafetyGateRef_A.RequestButton.Button
//     PlcTask Inputs/MAIN._Peripherie._Handling._components.SafetyGateRef_A.StartButton.Button <-> Channel 1/MAIN._Peripherie._Handling._components.SafetyGateRef_A.StartButton.Button
//   PLC/PLC Instance <-> Device 3 (EtherCAT)/Term 1 (EK1100)/Ovens (EK1122)/Oven_A (EK1100)/Term 15 (EL2004)
//     PlcTask Outputs/MAIN._Peripherie._Handling._components.SafetyGateRef_A.LockButton.Light <-> Channel 3/MAIN._Peripherie._Handling._components.SafetyGateRef_A.LockButton.Light
//     PlcTask Outputs/MAIN._Peripherie._Handling._components.SafetyGateRef_A.RequestButton.Light <-> Channel 2/MAIN._Peripherie._Handling._components.SafetyGateRef_A.RequestButton.Light
//     PlcTask Outputs/MAIN._Peripherie._Handling._components.SafetyGateRef_A.StartButton.Light <-> Channel 1/MAIN._Peripherie._Handling._components.SafetyGateRef_A.StartButton.Light
//   PLC/PLC Instance <-> Device 3 (EtherCAT)/Term 1 (EK1100)/Ovens (EK1122)/Oven_B (EK1100)/Term 22 (EL1004)
//     PlcTask Inputs/MAIN._Peripherie._Handling._components.SafetyGateRef_B.LockButton.Button <-> Channel 3/MAIN._Peripherie._Handling._components.SafetyGateRef_B.LockButton.Button
//     PlcTask Inputs/MAIN._Peripherie._Handling._components.SafetyGateRef_B.RequestButton.Button <-> Channel 2/MAIN._Peripherie._Handling._components.SafetyGateRef_B.RequestButton.Button
//     PlcTask Inputs/MAIN._Peripherie._Handling._components.SafetyGateRef_B.StartButton.Button <-> Channel 1/MAIN._Peripherie._Handling._components.SafetyGateRef_B.StartButton.Button
//   PLC/PLC Instance <-> Device 3 (EtherCAT)/Term 1 (EK1100)/Ovens (EK1122)/Oven_B (EK1100)/Term 23 (EL2004)
//     PlcTask Outputs/MAIN._Peripherie._Handling._components.SafetyGateRef_B.LockButton.Light <-> Channel 3/MAIN._Peripherie._Handling._components.SafetyGateRef_B.LockButton.Light
//     PlcTask Outputs/MAIN._Peripherie._Handling._components.SafetyGateRef_B.RequestButton.Light <-> Channel 2/MAIN._Peripherie._Handling._components.SafetyGateRef_B.RequestButton.Light
//     PlcTask Outputs/MAIN._Peripherie._Handling._components.SafetyGateRef_B.StartButton.Light <-> Channel 1/MAIN._Peripherie._Handling._components.SafetyGateRef_B.StartButton.Light
//   PLC/PLC Instance <-> Device 3 (EtherCAT)/Term 1 (EK1100)/Term 33 (EL6910)
//     PlcTask Inputs/MAIN._Peripherie._Handling._components.RackFeederRef.tsAckReq <-> StandardInputs/Rackfeeder_Axis.Error_AckReq_121
//     PlcTask Inputs/MAIN._Peripherie._Handling._components.RackFeederRef.tsSS1 <-> StandardInputs/Rackfeeder_Axis.SS1_Active_82
//     PlcTask Inputs/MAIN._Peripherie._Handling._components.RackFeederRef.tsSTO <-> StandardInputs/Rackfeeder_Axis.STO_Active_84
//     PlcTask Inputs/MAIN._Peripherie._Handling._components.SafetyGateRef_A.tsOpen <-> StandardInputs/SafetyGates.Open_A_75
//     PlcTask Inputs/MAIN._Peripherie._Handling._components.SafetyGateRef_A.tsSafe <-> StandardInputs/SafetyGates.Safe_A_73
//     PlcTask Inputs/MAIN._Peripherie._Handling._components.SafetyGateRef_B.tsOpen <-> StandardInputs/SafetyGates.Open_B_76
//     PlcTask Inputs/MAIN._Peripherie._Handling._components.SafetyGateRef_B.tsSafe <-> StandardInputs/SafetyGates.Safe_B_74
//     PlcTask Inputs/MAIN._Peripherie._Handling._components.SegmentDoorRef_A.tsAckReq <-> StandardInputs/Oven_Axis.Error_AckReq_OvenA_90
//     PlcTask Inputs/MAIN._Peripherie._Handling._components.SegmentDoorRef_A.tsSS1 <-> StandardInputs/Oven_Axis.SS1_Active_OvenA_92
//     PlcTask Inputs/MAIN._Peripherie._Handling._components.SegmentDoorRef_A.tsSTO <-> StandardInputs/Oven_Axis.STO_Active_OvenA_94
//     PlcTask Inputs/MAIN._Peripherie._Handling._components.SegmentDoorRef_B.tsAckReq <-> StandardInputs/Oven_Axis.Error_AckReq_OvenB_126
//     PlcTask Inputs/MAIN._Peripherie._Handling._components.SegmentDoorRef_B.tsSS1 <-> StandardInputs/Oven_Axis.SS1_Active_OvenB_125
//     PlcTask Inputs/MAIN._Peripherie._Handling._components.SegmentDoorRef_B.tsSTO <-> StandardInputs/Oven_Axis.STO_Active_OvenB_127
//     PlcTask Inputs/MAIN._Peripherie._Handling._components.TwinSAFERef.atsEmergencyActive[0] <-> StandardInputs/TwinSafeMain.Emergency01_Active_63
//     PlcTask Inputs/MAIN._Peripherie._Handling._components.TwinSAFERef.atsEmergencyActive[1] <-> StandardInputs/TwinSafeMain.Emergency02_Active_64
//     PlcTask Inputs/MAIN._Peripherie._Handling._components.TwinSAFERef.tsComErr <-> StandardInputs/TwinSafeMain.ComErr_99
//     PlcTask Inputs/MAIN._Peripherie._Handling._components.TwinSAFERef.tsEmergencySafe <-> StandardInputs/TwinSafeMain.Safe_62
//     PlcTask Inputs/MAIN._Peripherie._Handling._components.TwinSAFERef.tsFbErr <-> StandardInputs/TwinSafeMain.FBErr_98
//     PlcTask Inputs/MAIN._Peripherie._Handling._components.TwinSAFERef.tsFbRun <-> StandardInputs/TwinSafeMain.FBRun_100
//     PlcTask Inputs/MAIN._Peripherie._Handling._components.TwinSAFERef.tsInRun <-> StandardInputs/TwinSafeMain.InRun_55
//     PlcTask Inputs/MAIN._Peripherie._Handling._components.TwinSAFERef.tsOtherErr <-> StandardInputs/TwinSafeMain.OtherErr_56
//     PlcTask Inputs/MAIN._Peripherie._Handling._components.TwinSAFERef.tsOutErr <-> StandardInputs/TwinSafeMain.OutErr_101
//     PlcTask Outputs/MAIN._Peripherie._Handling._components.RackFeederRef.tsAck <-> StandardOutputs/Rackfeeder_Axis.Error_Ack_80
//     PlcTask Outputs/MAIN._Peripherie._Handling._components.SafetyGateRef_A.tsLockCmd <-> StandardOutputs/SafetyGates.LockCmd_A_109
//     PlcTask Outputs/MAIN._Peripherie._Handling._components.SafetyGateRef_A.tsRestart <-> StandardOutputs/SafetyGates.Restart_A_71
//     PlcTask Outputs/MAIN._Peripherie._Handling._components.SafetyGateRef_B.tsLockCmd <-> StandardOutputs/SafetyGates.LockCmd_B_110
//     PlcTask Outputs/MAIN._Peripherie._Handling._components.SafetyGateRef_B.tsRestart <-> StandardOutputs/SafetyGates.Restart_B_72
//     PlcTask Outputs/MAIN._Peripherie._Handling._components.SegmentDoorRef_A.tsAck <-> StandardOutputs/Oven_Axis.Error_Ack_OvenA_122
//     PlcTask Outputs/MAIN._Peripherie._Handling._components.SegmentDoorRef_B.tsAck <-> StandardOutputs/Oven_Axis.Error_Ack_OvenB_88
//     PlcTask Outputs/MAIN._Peripherie._Handling._components.TwinSAFERef.tsDriveRestart <-> StandardOutputs/TwinSafeMain.DriveRestart_117
//     PlcTask Outputs/MAIN._Peripherie._Handling._components.TwinSAFERef.tsEmergencyRestart <-> StandardOutputs/TwinSafeMain.Restart_61
//     PlcTask Outputs/MAIN._Peripherie._Handling._components.TwinSAFERef.tsErrAck <-> StandardOutputs/TwinSafeMain.ErrAck_53
//     PlcTask Outputs/MAIN._Peripherie._Handling._components.TwinSAFERef.tsRunStop <-> StandardOutputs/TwinSafeMain.RunStop_54
//   PLC/PLC Instance <-> NC-Task 1 SAF/Axes/Oven A
//     PlcTask Inputs/MAIN._Peripherie._Handling._components.SegmentDoorRef_A.VertikalAxis.NcToPlc <-> Outputs/ToPlc
//     PlcTask Outputs/MAIN._Peripherie._Handling._components.SegmentDoorRef_A.VertikalAxis.PlcToNc <-> Inputs/FromPlc
//   PLC/PLC Instance <-> NC-Task 1 SAF/Axes/Oven A CH1
//     PlcTask Inputs/MAIN._Peripherie._Handling._components.SegmentDoorRef_A.LatchLeft.NcToPlc <-> Outputs/ToPlc
//     PlcTask Outputs/MAIN._Peripherie._Handling._components.SegmentDoorRef_A.LatchLeft.PlcToNc <-> Inputs/FromPlc
//   PLC/PLC Instance <-> NC-Task 1 SAF/Axes/Oven A CH2
//     PlcTask Inputs/MAIN._Peripherie._Handling._components.SegmentDoorRef_A.LatchRight.NcToPlc <-> Outputs/ToPlc
//     PlcTask Outputs/MAIN._Peripherie._Handling._components.SegmentDoorRef_A.LatchRight.PlcToNc <-> Inputs/FromPlc
//   PLC/PLC Instance <-> NC-Task 1 SAF/Axes/Oven B
//     PlcTask Inputs/MAIN._Peripherie._Handling._components.SegmentDoorRef_B.VertikalAxis.NcToPlc <-> Outputs/ToPlc
//     PlcTask Outputs/MAIN._Peripherie._Handling._components.SegmentDoorRef_B.VertikalAxis.PlcToNc <-> Inputs/FromPlc
//   PLC/PLC Instance <-> NC-Task 1 SAF/Axes/Oven B CH1
//     PlcTask Inputs/MAIN._Peripherie._Handling._components.SegmentDoorRef_B.LatchLeft.NcToPlc <-> Outputs/ToPlc
//     PlcTask Outputs/MAIN._Peripherie._Handling._components.SegmentDoorRef_B.LatchLeft.PlcToNc <-> Inputs/FromPlc
//   PLC/PLC Instance <-> NC-Task 1 SAF/Axes/Oven B CH2
//     PlcTask Inputs/MAIN._Peripherie._Handling._components.SegmentDoorRef_B.LatchRight.NcToPlc <-> Outputs/ToPlc
//     PlcTask Outputs/MAIN._Peripherie._Handling._components.SegmentDoorRef_B.LatchRight.PlcToNc <-> Inputs/FromPlc
//   PLC/PLC Instance <-> NC-Task 1 SAF/Axes/Rackfeeder Teleskop
//     PlcTask Inputs/MAIN._Peripherie._Handling._components.RackFeederRef.TelescopeAxis.NcToPlc <-> Outputs/ToPlc
//     PlcTask Outputs/MAIN._Peripherie._Handling._components.RackFeederRef.TelescopeAxis.PlcToNc <-> Inputs/FromPlc
//   PLC/PLC Instance <-> NC-Task 1 SAF/Axes/Rackfeeder X
//     PlcTask Inputs/MAIN._Peripherie._Handling._components.RackFeederRef.HorizontalAxis.NcToPlc <-> Outputs/ToPlc
//     PlcTask Outputs/MAIN._Peripherie._Handling._components.RackFeederRef.HorizontalAxis.PlcToNc <-> Inputs/FromPlc
//   PLC/PLC Instance <-> NC-Task 1 SAF/Axes/Rackfeeder Y
//     PlcTask Inputs/MAIN._Peripherie._Handling._components.RackFeederRef.VerticalAxis.NcToPlc <-> Outputs/ToPlc
//     PlcTask Outputs/MAIN._Peripherie._Handling._components.RackFeederRef.VerticalAxis.PlcToNc <-> Inputs/FromPlc

// ---- Components/TcaCarrier/Structures/TcaCarrierStatus.TcDUT
TYPE TcaCarrierStatus :
STRUCT
	WorkpiecePlaces : INT; // starts with 1
	PrimaryWorkpieceStatus : eTcaWorkpiecePlaceProgress;
	SecondaryWorkpieceStatus : eTcaWorkpiecePlaceProgress;
	PrimaryWorkpieceStatusCount : INT;
	SecondaryWorkpieceStatusCount : INT;
	ArrayOfCarrierStatus : ARRAY[0..eTcaWorkpiecePlaceProgress.MAXSIZE] OF INT;
	ConfigError	: BOOL;
END_STRUCT
END_TYPE

// ---- Components/TcaPushButton/Structures/TcaPushButtonStatus.TcDUT
TYPE TcaPushButtonStatus :
STRUCT
	LightState : eTcaPushButtonLightState;
	Light : BOOL;	
	Signal : BOOL;
	Raising : BOOL;
	Falling : BOOL;
	ElapsedTime : TIME;
END_STRUCT
END_TYPE

// ---- Components/TcaPushButton/Structures/TcaPushButtonRef.TcDUT
TYPE TcaPushButtonRef :
STRUCT
	Button AT%I* : BOOL;
	Light AT%Q* : BOOL;	
END_STRUCT
END_TYPE

// ---- Components/TcaPushButton/Structures/TcaPushButtonConfig.TcDUT
TYPE TcaPushButtonConfig :
STRUCT
	LightState : eTcaPushButtonLightState;
	ButtonColor : eTcaPushButtonColor;
	ValidationTime	: TIME := T#100MS;
	FlashArray : ARRAY[0..128] OF TIME;
END_STRUCT
END_TYPE

// ---- Components/TcaStorage/E_ApproachDirection.TcDUT
{attribute 'qualified_only'}
TYPE E_ApproachDirection :
(
	Positive_X := 0,
	Positive_Y := 1,
	Positive_Z := 2,
	Negative_X := 3,
	Negative_Y := 4,
	Negative_Z := 5
);
END_TYPE

// ---- Components/TcaTrolley/TcaTrolleyRef.TcDUT
TYPE TcaTrolleyRef :
STRUCT
	Sensor AT%I* : BOOL;	
END_STRUCT
END_TYPE

// ---- Components/TcaWorkpiecePlace/Enumerations/eTcaWorkpiecePlaceProgress.TcDUT
{attribute 'qualified_only'}
{attribute 'strict'}
{attribute 'to_string'}
TYPE eTcaWorkpiecePlaceProgress :
(
	undefined := 0,
	blank,
	inProcess,
	finished,
	Error,
	
	MAXSIZE
);
END_TYPE

// ---- Components/TcaWorkpiecePlace/Enumerations/eTcaWorkpiecePlaceStatus.TcDUT
{attribute 'qualified_only'}
{attribute 'strict'}
{attribute 'to_string'}
TYPE eTcaWorkpiecePlaceStatus :
(
	undefined := 0,
	Ready,
	Prepared,
	Loaded,
	Locked,
	
	MAXSIZE
);
END_TYPE

// ---- Components/TcaWorkpiecePlace/Structures/TcaWorkpiecePlaceConfig.TcDUT
TYPE TcaWorkpiecePlaceConfig EXTENDS ST_ComboboxEntry:
STRUCT
	
END_STRUCT
END_TYPE

// ---- Components/TcaWorkpiecePlace/Structures/TcaWorkpiecePlaceStatus.TcDUT
TYPE TcaWorkpiecePlaceStatus : // EXTENDS ST_ComboboxEntry:
STRUCT
    ActionDescription : STRING(100);	
	Id : INT;
	Color: COLOR;
	PlaceStatus : eTcaWorkpiecePlaceStatus;
	Progress : eTcaWorkpiecePlaceProgress;
	
END_STRUCT
END_TYPE

// ---- Components_RMTH/TcaLaserDistanceSenor/Structures/TcaLaserDistanceSenorConfig.TcDUT
TYPE
    TcaLaserDistanceSenorConfig :
    STRUCT
        RawLow   : DINT;
        RawHigh  : DINT;
        RealLow  : REAL;
        RealHigh : REAL;
        Gain     : REAL := 1.0;
        Offset   : REAL := 0.0;
    END_STRUCT
END_TYPE

// ---- Components_RMTH/TcaLaserDistanceSenor/Structures/TcaLaserDistanceSenorStatus.TcDUT
(*~
<docu>
	<summary>
		`TcoAi` status structure.								
	</summary>				
</docu>	
~*)
TYPE
    TcaLaserDistanceSenorStatus :
    STRUCT
		{attribute addProperty Name "<#Raw range#>"}
        RawRange : REAL;
		{attribute addProperty Name "<#Real range#>"}
        RealRange : REAL;
		{attribute addProperty Name "<#Scaled value#>"}
        Scaled : REAL;
    END_STRUCT
END_TYPE

// ---- Components_RMTH/TcaLaserDistanceSenor/Structures/TcaLaserDistanceSenorService.TcDUT
TYPE TcaLaserDistanceSenorService :
STRUCT

END_STRUCT
END_TYPE

// ---- Components_RMTH/TcaRackFeeder/Structures/TcaRackFeederConfig.TcDUT
TYPE TcaRackFeederConfig :
STRUCT
END_STRUCT
END_TYPE

// ---- Components_RMTH/TcaRackFeeder/Structures/TcaRackFeederRef.TcDUT
TYPE TcaRackFeederRef :
STRUCT
	// Components
	VerticalAxis : TcoAxisRef;	
	HorizontalAxis: TcoAxisRef;
	TelescopeAxis : TcoAxisRef;
	
	// Sensor
	ReferenceSensor_Vertical AT%I* : BOOL;
	ReferenceSensor_Horizontal AT%I* : BOOL;
	ReferenceSensor_Telescope AT%I* : BOOL;
	
	// LaserDistanceSensor
	SensorLeftRef : TcaLaserDistanceSenorRef;	
	SensorRightRef : TcaLaserDistanceSenorRef;	
	
	// Safety
	tsSS1 AT%I* : BOOL;
	tsSTO AT%I* : BOOL;
	tsAckReq AT%I* : BOOL;
	tsAck AT%Q* : BOOL;
END_STRUCT
END_TYPE

// ---- Components_RMTH/TcaSafetyGate/Structures/TcaSafetyGateConfig.TcDUT
TYPE TcaSafetyGateConfig :
STRUCT
	
END_STRUCT
END_TYPE

// ---- Components_RMTH/TcaSegmentDoor/Structures/TcaSegmentDoorConfig.TcDUT
TYPE TcaSegmentDoorConfig :
STRUCT

END_STRUCT
END_TYPE

// ---- Components_RMTH/TcaSegmentDoor/Structures/TcaSegmentDoorStatus.TcDUT
TYPE TcaSegmentDoorStatus :
STRUCT
    ActionDescription : STRING(100);	         
	Safe : BOOL;
	Open : BOOL;
	
END_STRUCT
END_TYPE

// ---- Items/E_Coordinate.TcDUT
{attribute 'qualified_only'}
TYPE E_Coordinate :
(
	undefined := -1,
	x_axis := 0,
	y_axis := 1,
	z_axis := 2,
	u_axis := 3,
	v_axis := 4,
	w_axis := 5
);
END_TYPE

// ---- Items/ST_Coordinate.TcDUT
{attribute 'pack_mode' := '2'} 
TYPE ST_Coordinate :
STRUCT
	fX			: LREAL;
	fY			: LREAL;
	fZ			: LREAL;
	fRx			: LREAL;
	fRy			: LREAL;
	fRz			: LREAL;
	nOriginId	: INT;
END_STRUCT
END_TYPE

// ---- Template/Component_Cylinder/Structs/CylinderStatus.TcDUT
TYPE CylinderStatus :
STRUCT
	ActionDescription : STRING(100);	
END_STRUCT
END_TYPE

// ---- Template/RackFeeder/E_RackFeederCmd.TcDUT
{attribute 'qualified_only'}
{attribute 'strict'}
{attribute 'to_string'}
TYPE E_RackFeederCmd :
(
	noCmd := 0,
	TeachTrolleyDock,
	TeachStorageDock
);
END_TYPE

// ---- Template/RackFeeder/Structure/ST_StorageDock.TcDUT
TYPE ST_StorageDock :
STRUCT	
	sName				: STRING;
	nId					: INT;
	refStorage			: REFERENCE TO FB_Storage;
	posOrigin			: ST_Coordinate;
	bTeached			: BOOL;
	
END_STRUCT
END_TYPE

// ---- Template/RackFeeder/Structure/ST_TrolleyDock.TcDUT
TYPE ST_TrolleyDock :
STRUCT
	sName				: STRING;
	nId					: INT;
	refTrolley			: REFERENCE TO FB_Trolley;
	posButtom			: ST_Coordinate;
	posTop				: ST_Coordinate;
	bTeached			: BOOL;
	
END_STRUCT
END_TYPE

// ---- Template/Station/Data/ST001_ProcessData.TcDUT
TYPE ST001_ProcessData EXTENDS TcoData.TcoEntity:
STRUCT
	PressingTime : TIME;
END_STRUCT
END_TYPE

// ---- Template/Station/ST001_Components.TcDUT
TYPE ST001_Components : STRUCT
    PartPresent : TcoElements.TcoDi(MAIN_TECHNOLOGY._technology._ST001);
    StartButton : TcoElements.TcoDi(MAIN_TECHNOLOGY._technology._ST001);	
    Press : TcoPneumatics.TcoCylinder(MAIN_TECHNOLOGY._technology._ST001);	
	Drive : TcoDriveSimple(MAIN_TECHNOLOGY._technology._ST001);
END_STRUCT
END_TYPE

// ---- Utilities/Component/Enumerations/E_SafeState.TcDUT
{attribute 'qualified_only'}
{attribute 'strict'}
TYPE E_SafeState :
(
	None,
	Denied, 
	Permit
);
END_TYPE

// ---- Utilities/EventLog/Enumerations/E_BoolFilter.TcDUT
/// Listing of possible filter to a boolean variable
TYPE E_BoolFilter :
(
	eBoolFilter_none := 0,
	eBoolFilter_true,
	eBoolFilter_false
);
END_TYPE

// ---- Utilities/EventLog/Enumerations/E_FilterActive.TcDUT
/// enumeration of all possible priority
TYPE E_FilterActive :
(
	eFilter_none := 0,
	eFilter_activ := 1
);
END_TYPE

// ---- Utilities/EventLog/Enumerations/E_LogLevel.TcDUT
TYPE E_LogLevel :
(
	///kein Loglevel (nichts wird geloggt)
	eLogLevelNone := 0,
	///nur Fehler werden geloggt
	eLogLevelError := 1,
	///Fehler und Warnungen werden geloggt
	eLogLevelWarning := 2,
	///Fehler, Warnungen und Informationen werden geloggt
	eLogLevelInformation := 3
);
END_TYPE

// ---- Utilities/EventLog/Enumerations/ST_LoggingConfig.TcDUT
TYPE ST_LoggingConfig :
STRUCT
	/// <info>Angabe des Loggingproviders</info>
	eLoggingProvider: E_LoggingProvider;
	/// <info>Logging Name</info>
	sLogName: STRING;
	/// <info>Logging Pfad</info>
	sLogPath: STRING;
	/// <info>Logging Level</info>
	eLogLevel: E_LogLevel;
END_STRUCT
END_TYPE

// ---- Utilities/EventLog/Structures/ST_Event.TcDUT
/// Event structure
TYPE ST_Event EXTENDS ST_EventBase:
STRUCT
	dtRaiseTime			: DT;
	dtQuitTime			: DT;	
END_STRUCT
END_TYPE

// ---- Utilities/EventLog/Structures/ST_EventOutput.TcDUT
/// Event structure
TYPE ST_EventOutput :
STRUCT
	/// INDEX in global event-Array
	nIdx				: INT;		
	sPriority			: WSTRING;	
	nPriorityColor		: DWORD;
	sPosition			: T_MaxString;
	sDescription		: T_MaxString;
	sRaiseInfo			: STRING;

END_STRUCT
END_TYPE

// ---- Utilities/EventLog/Structures/ST_Log.TcDUT
TYPE ST_Log :
STRUCT
	sText: T_MaxString;
	sSource: STRING;
	bSaveRequest: BOOL;
	bSaved: BOOL;
	///	eLogLevelNone, eLogLevelError, eLogLevelWarning, eLogLevelInformation	
	eLevel: E_LogLevel;
	sTime: STRING;
END_STRUCT
END_TYPE

// ---- Utilities/EventLog/Visualization/Uc_EventLogControl.TcDUT
TYPE Uc_EventLogControl :
STRUCT	
	eAreaFilter 		: E_MachineArea := E_MachineArea.none;                   	
	bInfoFilter			: BOOL := TRUE;
	bWarningFilter		: BOOL := TRUE;
	bErrorFilter		: BOOL := TRUE;
		
	nErrorCount			: INT;
	nWarningCount		: INT;
	nInfoCount			: INT;
	
	bFilterChanged		: BOOL;
	
	nErrorColor			: DWORD;	
	nWarningColor		: DWORD;
	nInfoColor			: DWORD;
	
	bQuittAll			: BOOL;
	bMute				: BOOL;
	
	
END_STRUCT
END_TYPE

// ---- Utilities/EventLog/Visualization/Uc_EventLogTable.TcDUT
TYPE Uc_EventLogTable :
STRUCT
	astEvents			: ARRAY[0..nMaxEvents] OF ST_EventOutput;

	bQuitt				: BOOL;
	nIdx				: INT;	
	
	bAckn				: BOOL;
	bMute				: BOOL;
END_STRUCT
END_TYPE

// ---- Utilities/Helpers/Color/ST_Color.TcDUT
TYPE ST_Color :
STRUCT
	nTransparency				: BYTE;
	nRed						: BYTE;
	nGreen						: BYTE;
	nBlue						: BYTE;
END_STRUCT
END_TYPE

// ---- Utilities/List/Structures/Uc_List.TcDUT
TYPE Uc_List :
STRUCT
	nSelected			: UINT;
	ptSelected			: POINTER TO BYTE;
	astEntries			: ARRAY[0..255] OF ST_Listentry;
	bRemove				: BOOL;
	bInsert				: BOOL;
	bMoveUp				: BOOL;
	bMoveDown			: BOOL;
	bSave				: BOOL;
END_STRUCT
END_TYPE

// ---- Utilities/Sequencer/Enumeration/E_SequenceState.TcDUT
{attribute 'qualified_only'}
TYPE E_SequenceState :
(
	none := 0,		/// Status nicht gesetzt
	running,		/// Sequence läuft
	waiting,		/// Sequence wartet im Schritt
	finished,		/// Sequence fertig/ok
	error,			/// Sequence fehlgeschlagen
	error_running	/// Fehlerbehebung läuft
);
END_TYPE

// ---- Utilities/HexColor.TcGVL
VAR_GLOBAL
	
	textFontName		: STRING := 'Segoe UI Light';
	textH1				: INT := 26;
	textH2				: INT := 18;
	textH3				: INT := 10;
	colButton			: DWORD:=16#FFEBEBEB;
	colGrey01			: DWORD:=16#FFE3E3E3;
	colButtonHover		: DWORD:=colGrey01;
	colButtonDown		: DWORD:=16#FF9F9F9F;
	
	

	colSegmentReady 	:DWORD:=16#FF4D6C73;
	colSegmentLocked  	:DWORD:=16#FFA8BFB9;
	colSegmentError		:DWORD:=16#FFA64941;
	colSegmentWarning	:DWORD:=16#FFE4CE68;
	colSegmentFrame		:DWORD:=16#FF4D6C73;
	colSegmentSelect	:DWORD:=16#FFF2BE22;
	
	colSlotFrame		:DWORD:=16#FFB4BF5E;
	colSlotGlow			:DWORD:=16#FFDBF227;
	colSlotDisabled		:DWORD:=16#FFF3F5E6; //DCE0B8;
	colWhite 			:DWORD:=16#FFFFFFFF;
	
	colPmErrorFrame		:DWORD:=16#FF962B09;
	colPmOnFrame		:DWORD:=16#FFA66A75;
	colPmOffFrame		:DWORD:=16#FF9FA3A2;

	colPmErrorBg		:DWORD:=16#FFA64941;		
	colPmReadyBg		:DWORD:=16#FFF2F2F2;

	colHeatingOff		:DWORD:=16#FFA8BFB9;
	colHeatingDisconn	:DWORD:=16#FF0099DD;	
	colHeatingLow		:STRING:='FFF2BA52';
	colHeatingHigh		:STRING:='FFF24949';
	
	colStartButton		:DWORD:=16#FFE4CE68;
	colStopButton		:DWORD:=16#FFA64941;
	colWaitButton		:DWORD:=16#FF9FA3A2;
	
	colEventWarning		: DWORD := 16#FFF2B705;
	colEventInfo		: DWORD := 16#FF035AA6;
	colEventError		: DWORD := 16#FFD94032;
	colEventNone		: DWORD := 16#FF035AA6;
	
	
	colRibbon			:DWORD:=16#FF0099DD;
	colErrorBg			:DWORD:=16#FF9FA3A2;	
	
	colBlack 			: DWORD:=16#FF000000;
	colBlack00 			: DWORD:=16#00000000;
	colBlack25 			: DWORD:=16#40000000;
	colBlack50 			: DWORD:=16#80000000;
	colBlack75 			: DWORD:=16#C0000000;
	
	colLightRed			:DWORD:=16#FFD94032;
	colLightGreen		:DWORD:=16#FFB4BF5E;
	colLightBlue		:DWORD:=16#FF035AA6;
	colLightYellow		:DWORD:=16#FFF2B705;
	colLightGrey		:DWORD:=16#FFB2BEBF;
	colLightOrange		:DWORD:=16#FFF29F05;
	
	// COMP VISU
	// colCompErrorBg		:DWORD:=16#FFA64941;		
	// colCompReadyBg		:DWORD:=16#FFF2F2F2;	
	// colCompErrorFrame	:DWORD:=16#FF962B09;
	// colCompOnFrame		:DWORD:=16#FFA66A75;
	// colCompOffFrame		:DWORD:=16#FF9FA3A2;
	// colCompButton		:DWORD:=16#FF9FA3A2;
	// colCompButtonPush	:DWORD:=16#FF9FA3A2;
	
	
	colComp01			:DWORD:=16#FFF5D349;
	colComp02			:DWORD:=16#FF76A883;
	colComp03			:DWORD:=16#ffe0656b;
	colComp04			:DWORD:=16#FFCC9999;
	colCompBg			:DWORD:=16#FFF5F5F5;
	colCompSafe			:DWORD:=16#FFF5F5F5;
	colCompButton		:DWORD:=16#FFEBEBEB;
	
END_VAR

// ---- Utilities/Statics.TcGVL
VAR_GLOBAL
	/// current system time
	dtNow: DT;
	/// current system time in string format	
	sTimeString: STRING;
	/// PLC system informations
	stPlcSystemInfo: ST_PlcSystemInfo;
	/// default pulse struct
	stPulse: ST_DefaultPulse;
	/// logging buffer
	arLoggs: ARRAY[0..iLogArraySize] OF ST_Log;
	/// global stuff
	bForceStateChgAfterDrvReset: BOOL;
	bForcePreopBeforeDrvReset: BOOL;
	bLogDriveDiagMsgs: BOOL;
END_VAR

// ---- Template/Component_Cylinder/ITcoCylinder.TcIO
INTERFACE ITcoCylinder EXTENDS __System.IQueryInterface

PROPERTY AtHome : bool
GET
END_GET
END_PROPERTY

PROPERTY AtWork : bool
GET
END_GET
END_PROPERTY

METHOD MoveToHome : TcoCore.ITcoTaskStatus
END_METHOD

METHOD MoveToWork :TcoCore.ITcoTaskStatus
END_METHOD

(*~
	<docu>
		<summary>
			Stops cyclinder movement.
		 	<remarks>			
				<note type="important">
					This method switched off the signals for the movement of the piston in both direction.
					However depending on the pnemumatics configuration the movement may contintue if designed in that way.
					THIS IS NOT A SAFETY FUCTION!
				</note>
			</remarks>	 		
		</summary>			
	</docu>	
~*)
METHOD Stop : TcoCore.ITcoTaskStatus
END_METHOD

END_INTERFACE

// ---- Utilities/Component/Interfaces/ITF_Component.TcIO
INTERFACE ITF_Component EXTENDS __SYSTEM.IQueryInterface

PROPERTY AccessPermit : BOOL
GET
END_GET
END_PROPERTY

/// RunSuper component logic
{attribute 'object_name' := 'Base'}
METHOD Base
END_METHOD

PROPERTY BMK : STRING
GET
END_GET
SET
END_SET
END_PROPERTY

/// Get's or set's a value indicating whether this component is active or not.
PROPERTY Enable : BOOL
GET
END_GET
SET
END_SET
END_PROPERTY

/// Halt component logic
{attribute 'object_name' := 'Halt'}
METHOD Halt : E_OperationResult
VAR_INPUT
	StoppCategory					: INT;			// 0...ungesteuertes Stillsetzen     1...gesteuertes Stillsetzen     2...gesteuertes Stillsetzen ohne Trennung der Energiezufuhr							
END_VAR
END_METHOD

PROPERTY ID : INT
GET
END_GET
SET
END_SET
END_PROPERTY

/// Init component logic
{attribute 'object_name' := 'Init'}
METHOD Init : E_OperationResult
END_METHOD

PROPERTY MachineArea : E_MachineArea
GET
END_GET
SET
END_SET
END_PROPERTY

PROPERTY Name : STRING
GET
END_GET
SET
END_SET
END_PROPERTY

PROPERTY Path : String
GET
END_GET
END_PROPERTY

METHOD RegisterSafetyComp : BOOL
VAR_INPUT
	SafetyComp				: ITF_SafetyComp;
END_VAR
END_METHOD

/// Reset component logic
{attribute 'object_name' := 'Reset'}
METHOD Reset : E_OperationResult
END_METHOD

/// RestartSuper component logic
{attribute 'object_name' := 'Restart'}
METHOD Restart : E_OperationResult
VAR_INPUT
END_VAR
END_METHOD

/// Run component logic
{attribute 'object_name' := 'Run'}
METHOD Run
END_METHOD

PROPERTY SafeEnvironment : BOOL
GET
END_GET
END_PROPERTY

/// Get's value representing the component state.
PROPERTY State : E_ComponentState
GET
END_GET
END_PROPERTY

/// Get's value representing the component state.
PROPERTY StateAsString : STRING
GET
END_GET
END_PROPERTY

PROPERTY Typ : E_ComponentType
GET
END_GET
END_PROPERTY

END_INTERFACE

// ---- Utilities/EventLog/Interface/ITF_EventLog.TcIO
INTERFACE ITF_EventLog

/// sets the corresponding notification item flag raised
{attribute 'object_name' := 'SetEvent'}
METHOD SetEvent //: REFERENCE TO ST_Event
VAR_INPUT
	/// item to set
	stEvent			: ST_Event;
END_VAR
END_METHOD

END_INTERFACE

// ---- Components/TcaCarrier/Tasks/TcaCarrierModifyTask.TcPOU
FUNCTION_BLOCK TcaCarrierModifyTask EXTENDS TcoCore.TcoTask



VAR_IN_OUT
	inoArrayOfWorkpiecePlaces : ARRAY[*] OF TcaWorkpiecePlace(THIS^);	
END_VAR
VAR
    {attribute addProperty Name "<#Command#>"}
	_Command : eTcaCarrierCmd;
    {attribute addProperty Name "<#StatusOfWorkpiece#>"}
	_StatusOfWorkpiece : eTcaWorkpiecePlaceProgress;
	_StatusOfPlace : eTcaWorkpiecePlaceStatus;
    {attribute addProperty Name "<#CarrierConfig#>"}
	_CarrierConfig : TcaCarrierConfig;
END_VAR
VAR
    {attribute 'hide'}
	_WorkpiecePlaces : INT;
    {attribute 'hide'}
	_i	: DINT;
END_VAR

IF(Execute()) THEN	
	
	// Change of Config -> set to empty Place
	IF _Command = eTcaCarrierCmd.ConfigCarrier THEN
		Carrier.Config := _CarrierConfig;
		_Command := eTcaCarrierCmd.emptyPlaces;
		_StatusOfPlace := eTcaWorkpiecePlaceStatus.Ready;
		_StatusOfWorkpiece := eTcaWorkpiecePlaceProgress.blank;
	END_IF
	
	Carrier.RefreshStatus();
	_WorkpiecePlaces := Carrier.Status.WorkpiecePlaces;
	
	IF _WorkpiecePlaces = 0 THEN
		RETURN;
	END_IF

	CASE _Command OF	

	eTcaCarrierCmd.emptyPlaces : 
		FOR _i := LOWER_BOUND(inoArrayOfWorkpiecePlaces,1) TO UPPER_BOUND(inoArrayOfWorkpiecePlaces,1) DO
			inoArrayOfWorkpiecePlaces[_i].WorkpiecePresent := FALSE;
			inoArrayOfWorkpiecePlaces[_i].Status.PlaceStatus := _StatusOfPlace;
			inoArrayOfWorkpiecePlaces[_i].Status.Progress := _StatusOfWorkpiece;
			//inoArrayOfWorkpiecePlaces[_i].Id := TO_INT(_i)+1;
		END_FOR
		
		FOR _i := _WorkpiecePlaces TO UPPER_BOUND(inoArrayOfWorkpiecePlaces,1) DO
			inoArrayOfWorkpiecePlaces[_i].Restore();
			inoArrayOfWorkpiecePlaces[_i].Status.PlaceStatus := eTcaWorkpiecePlaceProgress.undefined;
			inoArrayOfWorkpiecePlaces[_i].Status.Progress := eTcaWorkpiecePlaceStatus.undefined;
			//inoArrayOfWorkpiecePlaces[_i].Id := -1;
		END_FOR
			

	eTcaCarrierCmd.fillPlaces : 
		FOR _i := LOWER_BOUND(inoArrayOfWorkpiecePlaces,1) TO _WorkpiecePlaces-1 DO
			inoArrayOfWorkpiecePlaces[_i].WorkpiecePresent := TRUE;
			inoArrayOfWorkpiecePlaces[_i].Status.PlaceStatus := _StatusOfPlace;
			inoArrayOfWorkpiecePlaces[_i].Status.Progress := _StatusOfWorkpiece;
			//inoArrayOfWorkpiecePlaces[_i].Id := TO_INT(_i)+1;
		END_FOR
		
		FOR _i := _WorkpiecePlaces TO UPPER_BOUND(inoArrayOfWorkpiecePlaces,1) DO
			inoArrayOfWorkpiecePlaces[_i].Restore();
			inoArrayOfWorkpiecePlaces[_i].Status.PlaceStatus := eTcaWorkpiecePlaceProgress.undefined;
			inoArrayOfWorkpiecePlaces[_i].Status.Progress := eTcaWorkpiecePlaceStatus.undefined;
			//inoArrayOfWorkpiecePlaces[_i].Id := -1;
		END_FOR
	
	eTcaCarrierCmd.RestorePlaces : 
		FOR _i := LOWER_BOUND(inoArrayOfWorkpiecePlaces,1) TO UPPER_BOUND(inoArrayOfWorkpiecePlaces,1) DO
			inoArrayOfWorkpiecePlaces[_i].Restore();
			//inoArrayOfWorkpiecePlaces[_i].Id := -1;
			inoArrayOfWorkpiecePlaces[_i].WorkpiecePresent := FALSE;
			inoArrayOfWorkpiecePlaces[_i].Status.PlaceStatus := eTcaWorkpiecePlaceProgress.blank;
			inoArrayOfWorkpiecePlaces[_i].Status.Progress := eTcaWorkpiecePlaceStatus.Ready;
		END_FOR

	END_CASE
	
	Carrier.RefreshStatus();
	DoneWhen(TRUE);
	Restore();
END_IF

PROPERTY Carrier : REFERENCE TO TcaCarrier
GET
VAR
    _carrier : POINTER TO TcaCarrier;
END_VAR
IF __QUERYPOINTER(_ParentObject,_carrier) THEN 	// Check if _Parent is Carrier
	Carrier REF= _carrier^;              		// If the check is successful dereference a pointer. simlar to THIS^ or SUPER^
END_IF
END_GET
END_PROPERTY

METHOD InvokeCarrierConfig : ITcoTaskStatus
VAR_INPUT
	inConfig : TcaCarrierConfig;
END_VAR
_CarrierConfig := inConfig;
InvokeCarrierConfig := This^.Invoke();
END_METHOD

METHOD InvokeWorkpieceCommand : ITcoTaskStatus
VAR_INPUT
	inCommand : eTcaCarrierCmd;
	inStatusOfWorkpiece : eTcaWorkpiecePlaceProgress;
END_VAR
_Command := inCommand;
_StatusOfWorkpiece := inStatusOfWorkpiece;
InvokeWorkpieceCommand := This^.Invoke();
END_METHOD

END_FUNCTION_BLOCK

// ---- Components/TcaCarrier/TcaCarrier.TcPOU
FUNCTION_BLOCK TcaCarrier EXTENDS TcoCore.TcoComponent IMPLEMENTS ITcaCarrier
VAR CONSTANT
	MAX_WORKPIECEPLACES : INT := 127;
END_VAR

VAR PERSISTENT
	_carrierID : INT;	
	_config : TcaCarrierConfig;
	_arrayOfWorkpiecePlaces : ARRAY[0..MAX_WORKPIECEPLACES] OF TcaWorkpiecePlace(THIS^);
END_VAR

VAR
	_ModifyTask : TcaCarrierModifyTask(THIS^);	
	_modifyId : INT := 0;
	_status : TcaCarrierStatus;
	_i : INT;
END_VAR

THIS^._ModifyTask(inoArrayOfWorkpiecePlaces := _arrayOfWorkpiecePlaces);

FOR _i:= 0 TO MAX_WORKPIECEPLACES DO
	_arrayOfWorkpiecePlaces[_i]();
END_FOR

METHOD ChangeConfig : ITcoTaskStatus 
VAR_INPUT
	inConfig : TcaCarrierConfig;
END_VAR
ChangeConfig := _ModifyTask.InvokeCarrierConfig(inConfig);
END_METHOD

PROPERTY Config : REFERENCE TO TcaCarrierConfig
GET
Config REF= _config;
END_GET
SET
_config := Config;
END_SET
END_PROPERTY

METHOD CoordinatesOf : ST_Coordinate
VAR_INPUT
	WorkpiecePlace		: INT;
END_VAR

VAR
	tmpConfig			: TcaCarrierConfig;
	
	tmpOffset 			: REAL;
	tmpOddRow			: INT;
	tmpEvenRow			: INT;
	tmpWorkpieceCount	: INT;
	
	tmpPos		 		: INT;
	tmpLoc		 		: INT;		
	tmpRow 				: INT;
	//tmpLvl				: INT;
	
	nRowNumber			: INT;
	nLocationNumber		: INT; 
	
	tmpCoordinate 		: ST_Coordinate;		
	
END_VAR
IF WorkpiecePlace = 0 OR WorkpiecePlace > Status.WorkpiecePlaces OR Status.ConfigError THEN
	RETURN;
END_IF

tmpConfig := _Config;

CASE tmpConfig.eConfiguration OF
	eTcaCarrierConfig.Layout1 : 
		tmpOffset := 0;
		tmpOddRow := tmpConfig.PositionsInRow;
        tmpEvenRow := tmpConfig.PositionsInRow;
        tmpWorkpieceCount := tmpConfig.PositionsInRow*tmpConfig.PositionsInColumn;
		
    eTcaCarrierConfig.Layout2 :
		tmpOffset := 0.5;
		tmpOddRow := tmpConfig.PositionsInRow;
		tmpEvenRow := tmpConfig.PositionsInRow;
        tmpWorkpieceCount := tmpConfig.PositionsInRow*tmpConfig.PositionsInColumn;
		 
    eTcaCarrierConfig.Layout3 :
		 tmpOffset := -0.5;
		 tmpOddRow := tmpConfig.PositionsInRow;
         tmpEvenRow := tmpConfig.PositionsInRow;
         tmpWorkpieceCount := tmpConfig.PositionsInRow*tmpConfig.PositionsInColumn;	
		 
	eTcaCarrierConfig.Layout4 :
		 tmpOffset := -0.5;
		 tmpOddRow := tmpConfig.PositionsInRow;
         tmpEvenRow := tmpConfig.PositionsInRow + 1;
         tmpWorkpieceCount := tmpConfig.PositionsInRow*tmpConfig.PositionsInColumn + tmpConfig.PositionsInColumn/2;
		
	eTcaCarrierConfig.Layout5 :
		 tmpOffset := 0.5;
		 tmpOddRow := tmpConfig.PositionsInRow;
         tmpEvenRow := tmpConfig.PositionsInRow - 1;
         tmpWorkpieceCount := tmpConfig.PositionsInRow*tmpConfig.PositionsInColumn - tmpConfig.PositionsInColumn/2;
		 
END_CASE

// Bestimmen des Reihen und Spaltenndex und der x und y-Koordinate
tmpPos := (WorkpiecePlace - 1) MOD tmpWorkpieceCount;
tmpRow := tmpPos/(tmpOddRow + tmpEvenRow);	
tmpLoc := tmpPos MOD (tmpOddRow + tmpEvenRow);
//tmpLvl := (Position - 1)/tmpWorkpieceCount;


IF tmpLoc >= tmpOddRow THEN
    // gerade Reihe
    nRowNumber := tmpRow*2 + 1;
    nLocationNumber := tmpLoc - tmpOddRow;
    tmpCoordinate.fX := tmpConfig.ColumnDistance*(nLocationNumber + tmpOffset);
    tmpCoordinate.fY := tmpConfig.RowDistance*nRowNumber;
ELSE
    // ungerade Reihe
    nRowNumber := tmpRow*2;
    nLocationNumber := tmpLoc;
    tmpCoordinate.fX := tmpConfig.ColumnDistance*nLocationNumber;
    tmpCoordinate.fY := tmpConfig.RowDistance*nRowNumber;
END_IF
		

//tmpCoordinate.fZ := tmpLvl*fLevelDistance;

// Koordinaten zurückgeben
tmpCoordinate.nOriginId := 0;
CoordinatesOf := tmpCoordinate;
END_METHOD

METHOD CountEmptyPlaces : INT

VAR
	tmp				: INT;
	ni				: INT;
END_VAR
CountEmptyPlaces := 0;

FOR ni := 0 TO Status.WorkpiecePlaces-1 DO
	
	IF _arrayOfWorkpiecePlaces[ni].Error THEN
		CONTINUE;
	END_IF

	IF _arrayOfWorkpiecePlaces[ni].Lock THEN
		CONTINUE;
	END_IF

	IF NOT _arrayOfWorkpiecePlaces[ni].WorkpiecePresent THEN
		tmp := tmp + 1;	
	END_IF

END_FOR

CountEmptyPlaces := tmp;
END_METHOD

METHOD CountPlacesByStatus : INT
VAR_INPUT
	nStatus			: INT;
END_VAR

VAR
	tmp				: INT;
	ni				: INT;
END_VAR
CountPlacesByStatus := 0;

FOR ni := 0 TO Status.WorkpiecePlaces-1 DO
	
	IF _arrayOfWorkpiecePlaces[ni].Error THEN
		CONTINUE;
	END_IF

	IF _arrayOfWorkpiecePlaces[ni].Lock THEN
		CONTINUE;
	END_IF

	IF _arrayOfWorkpiecePlaces[ni].Status.Progress = nStatus THEN
			tmp := tmp + 1;
	END_IF
	
END_FOR

CountPlacesByStatus := tmp;
END_METHOD

METHOD EmptyPlaces : ITcoTaskStatus
EmptyPlaces := _ModifyTask.InvokeWorkpieceCommand(eTcaCarrierCmd.emptyPlaces, eTcaWorkpiecePlaceProgress.blank);
END_METHOD

//FB_Init ist immer implizit verfügbar und wird primär für die Initialisierung verwendet.
//Der Rückgabewert wird nicht ausgewertet. Für gezielte Einflussnahme können Sie
//die Methoden explizit deklarieren und darin mit dem Standard-Initialisierungscode 
//zusätzlichen Code bereitstellen. Sie können den Rückgabewert auswerten.
METHOD FB_Init: BOOL
VAR_INPUT    
bInitRetains: BOOL; // TRUE: Die Retain-Variablen werden initialisiert (Reset warm / Reset kalt)    
bInCopyCode: BOOL;  // TRUE: Die Instanz wird danach in den Kopiercode kopiert (Online-Change)
ParentObject : ITcoObject;
END_VAR
VAR
	_i : INT;
END_VAR
FOR _i:= 0 TO MAX_WORKPIECEPLACES DO
	_arrayOfWorkpiecePlaces[_i].Id := _i+1;
END_FOR
END_METHOD

METHOD FillWithWorkpieces_CustomState : ITcoTaskStatus
VAR_INPUT
	Status		: eTcaWorkpiecePlaceProgress;
END_VAR
FillWithWorkpieces_CustomState := _ModifyTask.InvokeWorkpieceCommand(eTcaCarrierCmd.fillPlaces, Status);
END_METHOD

{attribute 'TcRpcEnable'}
METHOD FillWithWorkpieces_FinalState : ITcoTaskStatus
VAR_INPUT
END_VAR
IF Config.eFinalState = eTcaWorkpiecePlaceProgress.undefined THEN
	RETURN;
END_IF

FillWithWorkpieces_FinalState := _ModifyTask.InvokeWorkpieceCommand(eTcaCarrierCmd.fillPlaces, Config.eFinalState);
END_METHOD

METHOD FillWithWorkpieces_InitialState : ITcoTaskStatus
VAR_INPUT
END_VAR
IF Config.eFinalState = eTcaWorkpiecePlaceProgress.undefined THEN
	RETURN;
END_IF

FillWithWorkpieces_InitialState := _ModifyTask.InvokeWorkpieceCommand(eTcaCarrierCmd.fillPlaces, Config.eInitialState);
END_METHOD

PROPERTY FinalState : eTcaWorkpiecePlaceProgress
GET
FinalState := Config.eFinalState;
END_GET
SET
Config.eFinalState := FinalState;
END_SET
END_PROPERTY

METHOD FindPlace : REFERENCE TO TcaWorkpiecePlace //-1..no Position found

VAR_INPUT
	Status		: eTcaWorkpiecePlaceStatus;
END_VAR

VAR
	ni				: INT;
END_VAR
FindPlace REF= 0;
FOR ni := 0 TO THIS^.Status.WorkpiecePlaces-1 DO
	IF NOT _arrayOfWorkpiecePlaces[ni].Error 
	   AND NOT _arrayOfWorkpiecePlaces[ni].Lock 
       AND (_arrayOfWorkpiecePlaces[ni].Status.PlaceStatus = Status OR Status < eTcaWorkpiecePlaceStatus.undefined) THEN
	   
		FindPlace REF= _arrayOfWorkpiecePlaces[ni];
		EXIT;
		
	END_IF	
END_FOR
END_METHOD

METHOD GetPlaceReference : REFERENCE TO TcaWorkpiecePlace
VAR_INPUT
	nIndexNr		: INT;
END_VAR
IF nIndexNr < 0 OR nIndexNr > MAX_WORKPIECEPLACES THEN
	RETURN;
END_IF

GetPlaceReference REF= _arrayOfWorkpiecePlaces[nIndexNr];
END_METHOD

PROPERTY InitialState : eTcaWorkpiecePlaceProgress
GET
InitialState := Config.eInitialState;
END_GET
SET
Config.eInitialState := InitialState;
END_SET
END_PROPERTY

METHOD Layout : REFERENCE TO TcaCarrier
VAR_INPUT
	inLayout : eTcaCarrierConfig;
END_VAR
THIS^._config.eConfiguration:= inLayout;
Layout REF= THIS^;
END_METHOD

PROPERTY ModifyTask : TcoCore.ITcoTaskStatus
GET
ModifyTask := _ModifyTask;
END_GET
END_PROPERTY

METHOD PositionsInColumn : REFERENCE TO TcaCarrier
VAR_INPUT
	inPositionsInColumn : INT;
END_VAR
THIS^._config.PositionsInColumn:= inPositionsInColumn;
PositionsInColumn REF= THIS^;
END_METHOD

METHOD PositionsInRow : REFERENCE TO TcaCarrier
VAR_INPUT
	inPositionsInRow : INT;
END_VAR
THIS^._config.PositionsInRow:= inPositionsInRow;
PositionsInRow REF= THIS^;
END_METHOD

METHOD RefreshStatus : BOOL
VAR
	ni			: INT;
END_VAR
CASE _config.eConfiguration OF	
	eTcaCarrierConfig.Layout1 : _status.WorkpiecePlaces := _config.PositionsInRow*_config.PositionsInColumn;		
    eTcaCarrierConfig.Layout2 : _status.WorkpiecePlaces := _config.PositionsInRow*_config.PositionsInColumn;		 
    eTcaCarrierConfig.Layout3 : _status.WorkpiecePlaces := _config.PositionsInRow*_config.PositionsInColumn;		 
	eTcaCarrierConfig.Layout4 : _status.WorkpiecePlaces := _config.PositionsInRow*_config.PositionsInColumn + _config.PositionsInColumn/2;		
	eTcaCarrierConfig.Layout5 : _status.WorkpiecePlaces := _config.PositionsInRow*_config.PositionsInColumn - _config.PositionsInColumn/2;		
	ELSE
		 _status.WorkpiecePlaces := 0;
END_CASE

MEMSET(ADR(_status.ArrayOfCarrierStatus), 0, SIZEOF(_status.ArrayOfCarrierStatus));
_status.PrimaryWorkpieceStatus := 0;
_status.SecondaryWorkpieceStatus := 0;

FOR ni := 0 TO _status.WorkpiecePlaces DO
		
	IF _arrayOfWorkpiecePlaces[ni].Status.Progress = eTcaWorkpiecePlaceProgress.undefined THEN
		CONTINUE;
	END_IF

	_status.ArrayOfCarrierStatus[_arrayOfWorkpiecePlaces[ni].Status.Progress] := _status.ArrayOfCarrierStatus[_arrayOfWorkpiecePlaces[ni].Status.Progress] + 1;
	
	IF _status.ArrayOfCarrierStatus[_arrayOfWorkpiecePlaces[ni].Status.Progress] >= _status.ArrayOfCarrierStatus[_status.PrimaryWorkpieceStatus] THEN
		_status.SecondaryWorkpieceStatus := _status.PrimaryWorkpieceStatus;
		_status.PrimaryWorkpieceStatus := _arrayOfWorkpiecePlaces[ni].Status.Progress;
	END_IF


END_FOR

IF _status.PrimaryWorkpieceStatus = _status.SecondaryWorkpieceStatus THEN
	_status.SecondaryWorkpieceStatus := 0;
END_IF

_modifyId := _modifyId + 1;
END_METHOD

METHOD ResetPlaces : ITcoTaskStatus
ResetPlaces := _ModifyTask.InvokeWorkpieceCommand(eTcaCarrierCmd.fillPlaces, eTcaWorkpiecePlaceProgress.undefined);
END_METHOD

(*~
	<docu>
		<summary>
			Restores this instance to the Ready state. Can be called explicitly or from within one of the restore mechanisms.	
		</summary>			
	</docu>	
~*)
METHOD Restore : TcoCore.ITcoRestorable

VAR
	_i : INT;
END_VAR
FOR _i:= 0 TO MAX_WORKPIECEPLACES DO
	_arrayOfWorkpiecePlaces[_i].Restore();
END_FOR

RefreshStatus();
END_METHOD

(*~
	<docu>
		<summary>
		    Custom service (manual, maintenance) logic.
			This method must be implemented in derived class.
		</summary>			
	</docu>	
~*)
METHOD PROTECTED ServiceMode
VAR
	_i : INT;
END_VAR
FOR _i:= 0 TO MAX_WORKPIECEPLACES DO
	_arrayOfWorkpiecePlaces[_i].Service();
END_FOR
END_METHOD

PROPERTY Status : REFERENCE TO TcaCarrierStatus
GET
Status REF= _status;
END_GET
END_PROPERTY

PROPERTY Task : TcoCore.ITcoTask
GET
Task := _ModifyTask;
END_GET
END_PROPERTY

END_FUNCTION_BLOCK

// ---- Components/TcaStorage/TcaRobotStorage.TcPOU
FUNCTION_BLOCK TcaRobotStorage EXTENDS TcaStorage 

VAR	
	nOriginId			: INT := -1;	
	eApproachDirection	: E_ApproachDirection;
	stSupportPoint		: ST_Coordinate;
	sPose				: STRING;
	
	bCarrierTeached		: ARRAY[0..nMaxCarrierTypes] OF BOOL;
	aOffset				: ARRAY[0..nMaxCarrierTypes] OF ST_Coordinate;
END_VAR

PROPERTY ApproachDirection : E_ApproachDirection
GET
ApproachDirection := eApproachDirection;
END_GET
SET
eApproachDirection := ApproachDirection;
END_SET
END_PROPERTY

PROPERTY OriginId : INT
GET
OriginId := nOriginId;
END_GET
SET
nOriginId := OriginId;
END_SET
END_PROPERTY

PROPERTY Pose : STRING
GET
Pose := sPose;
END_GET
SET
sPose := Pose;
END_SET
END_PROPERTY

METHOD RobotCoordinatesOf : ST_Coordinate
VAR_INPUT
	Position			: INT;
END_VAR

VAR
	tmpCoordinate		: ST_Coordinate;
END_VAR
IF NOT bCarrierPresent OR NOT bCarrierTeached[_Carrier.CarrierId] OR nOriginId = -1 THEN
	RETURN;
END_IF

tmpCoordinate := _Carrier.CoordinatesOf(Position);

tmpCoordinate.nOriginId := nOriginId;
tmpCoordinate.fX := tmpCoordinate.fX + aOffset[_Carrier.CarrierId].fX;
tmpCoordinate.fY := tmpCoordinate.fY + aOffset[_Carrier.CarrierId].fY;
tmpCoordinate.fZ := tmpCoordinate.fZ + aOffset[_Carrier.CarrierId].fZ;
tmpCoordinate.fRx := tmpCoordinate.fRx + aOffset[_Carrier.CarrierId].fRx;
tmpCoordinate.fRy := tmpCoordinate.fRy + aOffset[_Carrier.CarrierId].fRy;
tmpCoordinate.fRz := tmpCoordinate.fRz + aOffset[_Carrier.CarrierId].fRz;

RobotCoordinatesOf := tmpCoordinate;
END_METHOD

PROPERTY SupportPoint : ST_Coordinate
GET
SupportPoint := stSupportPoint;
END_GET
SET
stSupportPoint := SupportPoint;
END_SET
END_PROPERTY

METHOD TeachCarrierType : TcoCore.ITcoTaskStatus
VAR_INPUT
	CarrierId					: INT;	
	Offset_X					: REAL;	
	Offset_Y					: REAL;	
	Offset_Z					: REAL;	
	Offset_Rx					: REAL;	
	Offset_Ry					: REAL;	
	Offset_Rz					: REAL;
END_VAR
aOffset[CarrierId].fX := Offset_X;
aOffset[CarrierId].fY := Offset_Y;
aOffset[CarrierId].fZ := Offset_Z;
aOffset[CarrierId].fRx := Offset_Rx;
aOffset[CarrierId].fRy := Offset_Ry;
aOffset[CarrierId].fRz := Offset_Rz;

bCarrierTeached[CarrierId] := TRUE;
END_METHOD

END_FUNCTION_BLOCK

// ---- Components/TcaTrolley/TcaTrolley.TcPOU
FUNCTION_BLOCK TcaTrolley EXTENDS TcoCore.TcoObject

VAR CONSTANT
	nMaxWorkpieceCarrier : INT := 31;
END_VAR

VAR_INPUT
	ref : REFERENCE TO TcaTrolleyRef;
END_VAR

VAR
	
	bDock					: BOOL;
	fbTrolleyPresent		: TcoDi(THIS^);	
	bTrolleyPresent			: BOOL;
	
	
	// Trolley Setting	
	nStoragePerRack			: INT;
	fStorageDivision		: LREAL;
	stOrigin				: ST_Coordinate; //mirrored for the Right side
	
	// Carrier Setting	
	fbCarrierTemplate		: TcaCarrier_(THIS^);	
	
END_VAR

VAR_OUTPUT PERSISTENT
	aLeftRack				: ARRAY[0..nMaxWorkpieceCarrier] OF TcaWorkpieceCarrier(THIS^);
	aRightRack				: ARRAY[0..nMaxWorkpieceCarrier] OF TcaWorkpieceCarrier(THIS^);
	bLeftRackPresent		: ARRAY[0..nMaxWorkpieceCarrier] OF BOOL;	
	bRightRackPresent		: ARRAY[0..nMaxWorkpieceCarrier] OF BOOL;	
END_VAR

VAR_INPUT
	cmd						: CMD_Trolley;
END_VAR

IF NOT __ISVALIDREF(ref) THEN
	bDock := FALSE;
ELSE
	bDock := TRUE;
	fbTrolleyPresent(inoSignal := ref.Sensor);
END_IF

METHOD AddCarrier : TcoCore.ITcoTaskStatus
VAR_IN_OUT
	WorkpieceCarrier			: TcaWorkpieceCarrier;
END_VAR
VAR_INPUT	
	bLeft						: BOOL;
	bRight						: BOOL;
	nId							: INT;
END_VAR
IF bLeft THEN
	MEMCPY(ADR(aLeftRack[nId]), ADR(WorkpieceCarrier), SIZEOF(TcaWorkpieceCarrier));
	bLeftRackPresent[nId] := TRUE;	
	aLeftRack[nId].RefreshCounter();
END_IF

IF bRight THEN
	MEMCPY(ADR(aRightRack[nId]), ADR(WorkpieceCarrier), SIZEOF(TcaWorkpieceCarrier));
	bRightRackPresent[nId] := TRUE;
	aRightRack[nId].RefreshCounter();
END_IF
END_METHOD

METHOD DefineCarrier
VAR_INPUT
	eConfiguration				: eTcaCarrierConfig;	
    nPosInRow					: INT;			// Numbers of Positions in first Row
    fRowDistance				: REAL;		// Distance from one Row to the other 
    nPosInColumn				: INT;			// Numbers of Positions in one Column
    fColumnDistance				: REAL;		// Distance from one Column to the other
END_VAR
fbCarrierTemplate.PositionInColumn :=	nPosInColumn;
fbCarrierTemplate.PositionInRow := nPosInRow;
fbCarrierTemplate.ColumnDistance := fColumnDistance;
fbCarrierTemplate.RowDistance := fRowDistance;
fbCarrierTemplate.Configuration := eConfiguration;
END_METHOD

METHOD DefineTrolley
VAR_INPUT
	StoragePerRack		: INT;
	StorageDivision		: LREAL;
	//Origin				: ST_Coordinate; //mirrored for the Right side
END_VAR
nStoragePerRack := StoragePerRack;
fStorageDivision := StorageDivision;
//stOrigin := Origin;
END_METHOD

METHOD EmptyCarrier : BOOL
VAR_INPUT
	bLeft			: BOOL;
	bRight			: BOOL;
	nState			: INT;
	nId				: INT;
END_VAR
IF bLeft THEN
	IF aLeftRack[nId].CarrierId = -1 THEN
		EmptyCarrier := TRUE;
	END_IF	

	aLeftRack[nId].LoadTemplate(fbCarrierTemplate);
	aLeftRack[nId].EmptyPlaces(nState);
	aLeftRack[nId].CarrierId := nId+1;
	aLeftRack[nId].RefreshCounter();
	bLeftRackPresent[nId] := FALSE;
END_IF

IF bRight THEN
	IF aRightRack[nId].CarrierId = -1 THEN
		EmptyCarrier := TRUE;
	END_IF	
	
	aRightRack[nId].LoadTemplate(fbCarrierTemplate);
	aRightRack[nId].EmptyPlaces(nState);
	aRightRack[nId].CarrierId := nId+1;
	aRightRack[nId].RefreshCounter();
	bRightRackPresent[nId] := FALSE;
END_IF
END_METHOD

METHOD EmptyTrolley : BOOL
VAR_INPUT
	bLeft			: BOOL;
	bRight			: BOOL;
END_VAR

VAR
	tmpNew			: BOOL;
	ni				: INT;
END_VAR
FOR ni:= 0 TO nMaxWorkpieceCarrier DO

	IF EmptyCarrier(bLeft, bRight, -1, ni) THEN
		tmpNew := TRUE;
	END_IF

END_FOR

IF tmpNew THEN
	ChangeToggle();
END_IF
END_METHOD

METHOD NewCarrier : BOOL
VAR_INPUT
	bLeft			: BOOL;
	bRight			: BOOL;
	nId				: INT;
	nState			: INT;
END_VAR
IF bLeft THEN
	IF aLeftRack[nId].CarrierId = -1 THEN
		NewCarrier := TRUE;
	END_IF

	aLeftRack[nId].LoadTemplate(fbCarrierTemplate);
	aLeftRack[nId].FillPlaces(nState);
	aLeftRack[nId].CarrierId := nId+1;
	aLeftRack[nId].RefreshCounter();
	bLeftRackPresent[nId] := TRUE;
END_IF

IF bRight THEN
	IF aRightRack[nId].CarrierId = -1 THEN
		NewCarrier := TRUE;
	END_IF	

	aRightRack[nId].LoadTemplate(fbCarrierTemplate);
	aRightRack[nId].FillPlaces(nState);
	aRightRack[nId].CarrierId := nId+1;
	aRightRack[nId].RefreshCounter();
	bRightRackPresent[nId] := TRUE;
END_IF
END_METHOD

METHOD NewTrolley : BOOL
VAR_INPUT
	bLeft			: BOOL;
	bRight			: BOOL;
	nState			: INT;
END_VAR

VAR
	tmpNew			: BOOL;
	ni				: INT;
END_VAR
FOR ni:= 0 TO nMaxWorkpieceCarrier DO

	IF NewCarrier(bLeft, bRight, ni, nState) THEN
		tmpNew := TRUE;
	END_IF
	
END_FOR

IF tmpNew THEN
	ChangeToggle();
END_IF
END_METHOD

METHOD RefreshTrolley
VAR
	ni	: INT;
END_VAR
FOR ni:= 0 TO nMaxWorkpieceCarrier DO
	aLeftRack[ni].RefreshCounter();
	aRightRack[ni].RefreshCounter();
END_FOR
END_METHOD

METHOD RemoveCarrier : TcoCore.ITcoTaskStatus
VAR_INPUT
	bLeft			: BOOL;
	bRight			: BOOL;
	nId				: INT;
END_VAR
IF bLeft THEN
	aLeftRack[nId].ResetPlaces();
	aLeftRack[nId].CarrierId := -1;
	bLeftRackPresent[nId] := FALSE;
	aLeftRack[nId].RefreshCounter();
END_IF

IF bRight THEN
	aRightRack[nId].ResetPlaces();
	aRightRack[nId].CarrierId := -1;
	bRightRackPresent[nId] := FALSE;
	aRightRack[nId].RefreshCounter();
END_IF
END_METHOD

METHOD RemoveTrolley : BOOL
VAR_INPUT
	bLeft			: BOOL;
	bRight			: BOOL;
END_VAR

VAR
	ni				: INT;
END_VAR
FOR ni:= 0 TO nMaxWorkpieceCarrier DO

	RemoveCarrier(bLeft, bRight, ni);

END_FOR

ChangeToggle();
END_METHOD

(*~
	<docu>
		<summary>
			Restores this instance to the Ready state. Can be called explicitly or from within one of the restore mechanisms.	
		</summary>			
	</docu>	
~*)
METHOD Restore : TcoCore.ITcoRestorable
END_METHOD

/// RunSuper component logic
{attribute 'object_name' := 'Run'}
METHOD  Run
END_METHOD

(*~
	<docu>
		<summary>
		    Custom service (manual, maintenance) logic.
			This method must be implemented in derived class.
		</summary>			
	</docu>	
~*)
METHOD PROTECTED ServiceMode
END_METHOD

/// Visu component logic
{attribute 'object_name' := 'Visu'}
METHOD  Visu

VAR
	ni			:INT;
END_VAR
CASE cmd.cmd OF
	eTcaTrolleyCmd.FillTrolley:
		NewTrolley(TRUE, TRUE, cmd.nId);
	
	eTcaTrolleyCmd.EmptyTrolley:
		EmptyTrolley(TRUE, TRUE);
	
	eTcaTrolleyCmd.RemoveTrolley:
		RemoveTrolley(TRUE, TRUE);
		
END_CASE

IF cmd.cmd <> eTcaTrolleyCmd.noCmd THEN
	cmd.cmd := eTcaTrolleyCmd.noCmd; 
END_IF

FOR ni:= 0 TO nMaxWorkpieceCarrier DO
	IF aLeftRack[ni].Cmd = eTcaCarrierCmd.changeState THEN
		NewCarrier(TRUE, FALSE, ni, cmd.nId);
		aLeftRack[ni].Cmd := eTcaCarrierCmd.noCmd;
	END_IF
	
	IF aRightRack[ni].Cmd = eTcaCarrierCmd.changeState THEN
		NewCarrier(FALSE, TRUE, ni, cmd.nId);
		aRightRack[ni].Cmd := eTcaCarrierCmd.noCmd;
	END_IF
	
END_FOR
END_METHOD

END_FUNCTION_BLOCK

// ---- Components_RMTH/TcaLaserDistanceSenor/TcaLaserDistanceSenor.TcPOU
FUNCTION_BLOCK TcaLaserDistanceSenor EXTENDS TcoCore.TcoComponent
VAR CONSTANT
	_dataArraylength : INT := 127;
END_VAR

VAR_INPUT
	ref : REFERENCE TO TcaLaserDistanceSenorRef;
END_VAR

VAR	
	
	_status : TcaLaserDistanceSenorStatus;
	_config : TcaLaserDistanceSenorConfig;
	_service : TcaLaserDistanceSenorService;
	
    _signalRef : REFERENCE TO TcaLaserDistanceSenorRef;
	_externalXSignal : REFERENCE TO DINT;
    _recordDataTask : TcoCore.TcoTask(THIS^);	
	_signal : DINT;	
	_signalInfo : TcoCore.TcoSignalInfo;
	_curveSketcher : FB_ALY_CurveSketcher_1Ch; 
	_recordtime	: TIME := T#50S;
	_recordintervall : TIME := T#200MS;
	_stopRecord	: BOOL;
	_PeakCount : INT := 0;	
	_ValleyCount : INT := 0;
	_DistanceCount : INT := 0;
	_ValleyArray : ARRAY[0.._dataArraylength] OF TcaLaserDistanceSensorDataArrayEntry;
	_PeakArray : ARRAY[0.._dataArraylength] OF TcaLaserDistanceSensorDataArrayEntry;	
	_DistanceArray : ARRAY[0.._dataArraylength] OF TcaLaserDistanceSensorDataArrayEntry;	
	_SumDistance : DINT;
	_MaxDistance : TcaLaserDistanceSensorDataArrayEntry;
	_MinDistance : TcaLaserDistanceSensorDataArrayEntry;	
END_VAR

IF NOT __ISVALIDREF(ref)  THEN
    Messenger.Post('<#Invalid reference signal #>', TcoCore.eMessageCategory.ProgrammingError);
    RETURN;
END_IF

_signalRef REF= ref;

// Signal Postprocessing
_signalInfo.GetSignalInfo(SIZEOF(_signalRef), ADR(_signalRef));
_signal := MIN(MAX(0,(_signalRef.Sensor/100)*100), 350000);


// Tasks
RecordDataTask();

PROPERTY AvgDistance : LREAL
GET
AvgDistance := _SumDistance/_DistanceCount;
END_GET
END_PROPERTY

PROPERTY Config : REFERENCE TO TcaLaserDistanceSenorConfig
GET
Config REF= _config;
END_GET
END_PROPERTY

PROPERTY FirstPeak : TcaLaserDistanceSensorDataArrayEntry
GET
FirstPeak := _PeakArray[0];
END_GET
END_PROPERTY

PROPERTY FirstValley : TcaLaserDistanceSensorDataArrayEntry
GET
FirstValley := _ValleyArray[0];
END_GET
END_PROPERTY

METHOD insideArea : BOOL
VAR_INPUT
	lowLimit			: DINT;
	highLimit			: DINT;
END_VAR
insideArea := _signal < highLimit AND _signal > lowLimit;
END_METHOD

METHOD isValue : BOOL
VAR_INPUT
	Value			: DINT;
	Epsilon			: DINT := 1000;
END_VAR
isValue := insideArea(Value-Epsilon, Value+Epsilon);
END_METHOD

PROPERTY MaxDistance : TcaLaserDistanceSensorDataArrayEntry
GET
MaxDistance := _MaxDistance;
END_GET
END_PROPERTY

PROPERTY MinDistance : TcaLaserDistanceSensorDataArrayEntry
GET
MinDistance := _MinDistance;
END_GET
END_PROPERTY

METHOD RecordData : TcoCore.ITcoTaskStatus
VAR_INPUT
	Recordtime			: TIME;
	RecordIntervall		: TIME;
END_VAR
RecordData := _recordDataTask.Invoke();
END_METHOD

METHOD RecordDataTask : BOOL
VAR	
	tmpX 		: DINT;
END_VAR
_recordDataTask.Enabled := TRUE;
_recordDataTask.Execute();

IF _recordDataTask.State = eTaskState.Ready THEN
	;
END_IF


IF _recordDataTask.State = eTaskState.Done OR _recordDataTask.Done THEN
	;
END_IF


IF _recordDataTask.State = eTaskState.Error THEN
	;
END_IF

// First STEP - Settings - Requested State was not possible
IF _recordDataTask.ElapsedTime = T#0MS THEN
	_curveSketcher.Reset();
	_curveSketcher.Configure(10000, TRUE, 1000);
	
	MEMSET(ADR(_PeakArray), 0, SIZEOF(_PeakArray));
	MEMSET(ADR(_ValleyArray), 0, SIZEOF(_ValleyArray));
	MEMSET(ADR(_MaxDistance), 0, SIZEOF(_MaxDistance));
	MEMSET(ADR(_MinDistance), 0, SIZEOF(_MinDistance));
	_PeakCount := 0;	
	_ValleyCount := 0;
	_DistanceCount := 0;
END_IF

IF NOT _recordDataTask.Busy THEN
	RETURN;
END_IF

// Write Senor value into Array
_curveSketcher.SetChannelValue(_signal);
_curveSketcher.Call(TIME_TO_ULINT(_recordDataTask.ElapsedTime));

IF __ISVALIDREF(_externalXSignal) THEN
	tmpX := _externalXSignal;
ELSE
	tmpX := TIME_TO_DINT(_recordDataTask.ElapsedTime);	
END_IF
	
IF  ULINT_TO_INT(_curveSketcher.nCountPeaks) > _PeakCount THEN
	_PeakArray[_PeakCount].x := tmpX;	
	_PeakArray[_PeakCount].y := LREAL_TO_DINT(_curveSketcher.fLastPeak);
	_PeakCount := ULINT_TO_INT(_curveSketcher.nCountPeaks);
END_IF

IF ULINT_TO_INT(_curveSketcher.nCountValleys) > _ValleyCount THEN
	_ValleyArray[_ValleyCount].x := tmpX;	
	_ValleyArray[_ValleyCount].y := LREAL_TO_DINT(_curveSketcher.fLastValley);
	_ValleyCount := ULINT_TO_INT(_curveSketcher.nCountValleys);
END_IF

IF  _PeakCount - _ValleyCount > 0 AND (TIME_TO_DINT(_recordDataTask.ElapsedTime) MOD TIME_TO_DINT(_recordintervall)) = 0 THEN
	_DistanceArray[_DistanceCount].x := tmpX;
	_DistanceArray[_DistanceCount].y := _signal;
	
	IF _MinDistance.y > _signal THEN
		_MinDistance := _DistanceArray[_DistanceCount];
	END_IF
	
	IF _MaxDistance.y < _signal THEN
		_MaxDistance := _DistanceArray[_DistanceCount];
	END_IF
	
	_SumDistance := _SumDistance + _signal;			// during the Measurement sum of all Signals
	_DistanceCount := _DistanceCount + 1;
END_IF
	
IF _DistanceCount > _dataArraylength THEN
	_recordDataTask.Abort();
	_recordDataTask.Messenger.Error('Data Overflow');
END_IF

IF _PeakCount > _dataArraylength THEN
	_recordDataTask.Abort();
	_recordDataTask.Messenger.Error('Data Overflow');
END_IF

IF _ValleyCount > _dataArraylength THEN
	_recordDataTask.Abort();
	_recordDataTask.Messenger.Error('Data Overflow');
END_IF

	
// Task Done	
_recordDataTask.DoneWhen(_stopRecord);
_stopRecord := FALSE;
END_METHOD

(*~
	<docu>
		<summary>
			Restores this instance to the Ready state. Can be called explicitly or from within one of the restore mechanisms.	
		</summary>			
	</docu>	
~*)
METHOD  Restore : ITcoRestorable
// No implementation needed for this componet.
END_METHOD

(*~
	<docu>
		<summary>
		    Custom service (manual, maintenance) logic.
			This method must be implemented in derived class.
		</summary>			
	</docu>	
~*)
METHOD PROTECTED  ServiceMode
END_METHOD

PROPERTY SetExternalXSignal : DINT
SET
_externalXSignal REF= SetExternalXSignal;
END_SET
END_PROPERTY

PROPERTY Status : REFERENCE TO TcaLaserDistanceSenorStatus
GET
Status REF= _status;
END_GET
END_PROPERTY

METHOD StopRecordData
VAR_INPUT
END_VAR
_stopRecord := TRUE;
END_METHOD

END_FUNCTION_BLOCK

// ---- Components_RMTH/TcaRackFeeder/TcaRackFeeder.TcPOU
FUNCTION_BLOCK TcaRackFeeder EXTENDS TcoCore.TcoComponent

VAR_INPUT
	ref : REFERENCE TO TcaRackFeederRef;
END_VAR

VAR
	_status : TcaRackFeederStatus;
	_config : TcaRackFeederConfig;
	_service : TcaRackFeederService;
	
	_EnableAxis : BOOL := TRUE;
	_EnableAxisSafe : BOOL;	
	
	// Components
	_vertikalAxis : TcoDriveSimple(THIS^);	
	_horizontalAxis : TcoDriveSimple(THIS^);
	_telescopeAxis : TcoDriveSimple(THIS^);
	
END_VAR

IF NOT __ISVALIDREF(ref)  THEN
    Messenger.Post('<#Invalid reference signal #>', TcoCore.eMessageCategory.ProgrammingError);
    RETURN;
END_IF

// Axis
_EnableAxisSafe := _EnableAxis; //AND ref.tsSS1;
_vertikalAxis(inCalibrationCam:= ref.ReferenceSensor_Vertical, inEnable:=  _EnableAxisSafe , inEnableNegative:= _EnableAxisSafe, inEnablePositive:= _EnableAxisSafe, inoAxisRef:= ref.VerticalAxis);
_horizontalAxis(inCalibrationCam:= ref.ReferenceSensor_Horizontal, inEnable:=  _EnableAxisSafe , inEnableNegative:= _EnableAxisSafe, inEnablePositive:= _EnableAxisSafe, inoAxisRef:= ref.HorizontalAxis);
_telescopeAxis(inCalibrationCam:= ref.ReferenceSensor_Telescope, inEnable:=  _EnableAxisSafe , inEnableNegative:= _EnableAxisSafe, inEnablePositive:= _EnableAxisSafe, inoAxisRef:= ref.TelescopeAxis);

PROPERTY Config : REFERENCE TO TcaRackFeederConfig
GET
Config Ref= _config;
END_GET
SET
_config := Config;
END_SET
END_PROPERTY

METHOD DropCarrier : BOOL
VAR_INPUT
END_VAR
END_METHOD

METHOD FetchCarrier : BOOL
VAR_INPUT
END_VAR
END_METHOD

METHOD FindCarrier
VAR_INPUT
END_VAR
END_METHOD

{warning 'Methodenimplementierung hinzufügen'}
METHOD Restore : TcoCore.ITcoRestorable
END_METHOD

{warning 'Methodenimplementierung hinzufügen'}
(*~
	<docu>
		<summary>
		    Custom service (manual, maintenance) logic.
			This method must be implemented in derived class.
		</summary>			
	</docu>	
~*)
METHOD PROTECTED ServiceMode
END_METHOD

PROPERTY Status : REFERENCE TO TcaRackFeederStatus
GET
Status REF= _status;
END_GET
END_PROPERTY

METHOD TeachStorageBase
VAR_IN_OUT
END_VAR
END_METHOD

METHOD TeachTrolleyBase
VAR_IN_OUT
END_VAR
END_METHOD

END_FUNCTION_BLOCK

// ---- Components_RMTH/TcaTwinSAFE/TcaTwinSAFE.TcPOU
FUNCTION_BLOCK TcaTwinSAFE EXTENDS TcoComponent

VAR CONSTANT
	MAX_EMEGENCY	: INT := 2;
END_VAR

VAR_INPUT
	ref : REFERENCE TO TcaTwinSAFERef;
END_VAR

VAR
	_status : TcaTwinSAFEStatus;
	_config : TcaTwinSAFEConfig;
	_service : TcaTwinSAFEService;	

	_quittButton : TcaPushButton(THIS^);
	_ackTask : TcoTask(THIS^);
	_runTask : TcoTask(THIS^);
END_VAR

//RETURN;

IF NOT __ISVALIDREF(ref)  THEN
    Messenger.Post('<#Invalid reference signal #>', TcoCore.eMessageCategory.ProgrammingError);
    RETURN;
END_IF

// Button
_quittButton(ref:= ref.QuittButton);

// Task
_ackTask.Enabled := TRUE;
IF (_ackTask.Execute()) THEN	
	ref.tsRunStop := TRUE;

	IF NOT ref.tsFbRun THEN
		RETURN;
	END_IF
		
	// Twinsafe group Error
	IF CheckError() AND NOT ref.tsErrAck THEN
		ref.tsErrAck := TRUE;
	ELSE
		ref.tsErrAck := FALSE;
	END_IF

	// Emergency Restart
	IF NOT ref.tsEmergencySafe AND NOT ref.tsEmergencyRestart THEN
		ref.tsErrAck := TRUE;
		ref.tsEmergencyRestart := TRUE;	
	ELSE
		ref.tsErrAck := FALSE;
		ref.tsEmergencyRestart := FALSE;
	END_IF

	IF ref.tsInRun AND ref.tsEmergencySafe THEN	
		_ackTask.ThrowWhen(TRUE);
		_runTask.Restore();
		_runTask.Invoke();
	END_IF
END_IF

_runTask.Enabled := TRUE;
IF (_runTask.Execute()) THEN	
	_runTask.ThrowWhen(CheckError());	
END_IF

// Refresh Status
_status.Safe := ref.tsEmergencySafe; // todo components
_status.Error := CheckError();
_status.Running := ref.tsInRun AND ref.tsFbRun;
THIS^.Status;

METHOD Acknowledge : ITcoTaskStatus
VAR_INPUT
END_VAR
_ackTask.Restore();
Acknowledge := _ackTask.Invoke();
END_METHOD

PROPERTY AckTask : TcoCore.ITcoTask
GET
AckTask := _AckTask;
END_GET
END_PROPERTY

METHOD CheckError : BOOL
VAR
END_VAR
CheckError := FALSE;

IF ref.tsComErr THEN
	Messenger.Error('TwinSAFE COM Error');
	CheckError := TRUE;
END_IF

IF ref.tsFbErr THEN
	Messenger.Error('TwinSAFE FB Error');
	CheckError := TRUE;
END_IF		

IF ref.tsOutErr THEN
	Messenger.Error('TwinSAFE Out Error');
	CheckError := TRUE;
END_IF		

IF ref.tsOtherErr THEN
	Messenger.Error('TwinSAFE Other Error');
	CheckError := TRUE;
END_IF
END_METHOD

PROPERTY Config : REFERENCE TO TcaTwinSAFEConfig
GET
Config Ref= _config;
END_GET
SET
_config := Config;
END_SET
END_PROPERTY

{warning 'Methodenimplementierung hinzufügen'}
METHOD Restore : TcoCore.ITcoRestorable
Acknowledge();
END_METHOD

PROPERTY RunTask : TcoCore.ITcoTask
GET
RunTask := _RunTask;
END_GET
END_PROPERTY

{warning 'Methodenimplementierung hinzufügen'}
(*~
	<docu>
		<summary>
		    Custom service (manual, maintenance) logic.
			This method must be implemented in derived class.
		</summary>			
	</docu>	
~*)
METHOD PROTECTED ServiceMode
IF _quittButton.Status.Raising OR _service.QuittButton.Button THEN 
	_service.QuittButton.Button := FALSE;
	Acknowledge(); 
END_IF
END_METHOD

PROPERTY Status : REFERENCE TO TcaTwinSAFEStatus
GET
Status REF= _status;

_service.Error := status.Error;
_service.Running := status.Running;
_service.Safe := status.Safe;
END_GET
END_PROPERTY

END_FUNCTION_BLOCK

// ---- Program/Handling/Sequences/Handling_Teach.TcPOU
FUNCTION_BLOCK Handling_Teach EXTENDS TcoCore.TcoSequencer
VAR
	_o : TcoCore.TcoSequencerObserver(THIS^);	
	_dialog : TcoCore.TcoDialog(THIS^);
END_VAR

PROPERTY Components : REFERENCE TO Handling_Components
GET
VAR
    _parent : POINTER TO Handling;
END_VAR
IF __QUERYPOINTER(_ParentObject,_parent) THEN // Check if _Parent is Station001
	Components REF= _parent^._components;              // If the check is successful dereference a pointer. simlar to THIS^ or SUPER^
END_IF
END_GET
END_PROPERTY

(*~
	<docu>
		<summary>
			Main method of the sequener. Custom code needs to be placed here. The sequencer is executed by call of InstanceName.Run() method.
			This method is abstract, and it must be overridden in derived block.
		</summary>
	</docu>
~*)
METHOD PROTECTED  Main : BOOL
VAR
	test: TcEventEntry;
	answer : TcoCore.eCustomizedDialogAnswer;
	_answer: STRING(INT#3);
END_VAR
THIS^.Observer := _o;

IF (Step(0, TRUE, 'MOVE HORIZONTAL TO LOAD')) THEN
    //--------------------------------------------
	
	_dialog.Show()
			.WithType(eDialogType.Question)				
			.WithCaption('Ready to go?')
			.WithText('Do you really want to start movements? Do we go ahead?')			
			.WithYesNo();
			
	
	IF(_dialog.Answer = TcoCore.eDialogAnswer.Yes) THEN RequestStep(100); _dialog.Restore(); END_IF;
    IF(_dialog.Answer = TcoCore.eDialogAnswer.No) THEN RequestStep(200); _dialog.Restore(); END_IF;
	
    //StepCompleteWhen(_StepElapsedTime > T#5S);
    //--------------------------------------------	
END_IF;


IF (Step(100, TRUE, 'YEEEEEEES')) THEN
    //--------------------------------------------	
    StepCompleteWhen(_StepElapsedTime > T#10S);
    //--------------------------------------------		
END_IF;

IF (Step(200, TRUE, 'NOOOOOOO')) THEN
    //--------------------------------------------	
    StepCompleteWhen(_StepElapsedTime > T#10S);
    //--------------------------------------------		
END_IF;


IF (Step(300, TRUE, 'GROUND MODE COMPLETE')) THEN
    //--------------------------------------------
    //--------------------------------------------	
END_IF;
END_METHOD

END_FUNCTION_BLOCK

// ---- Program/Handling/Handling_Components.TcPOU
FUNCTION_BLOCK Handling_Components EXTENDS TcoCore.TcoObject 
VAR	
	// Safety
	_TwinSAFE : TcaTwinSAFE(THIS^);
	TwinSAFERef : TcaTwinSAFERef;
	
	_safetyGate_A : TcaSafetyGate(THIS^);
	SafetyGateRef_A : TcaSafetyGateRef;
	
	_safetyGate_B : TcaSafetyGate(THIS^);
	SafetyGateRef_B : TcaSafetyGateRef;


	// SegmentDoor
	_segmentDoor_A : TcaSegmentDoor(THIS^);
	SegmentDoorRef_A : TcaSegmentDoorRef;

	_segmentDoor_B : TcaSegmentDoor(THIS^);
	SegmentDoorRef_B : TcaSegmentDoorRef;	
	
	
	// RackFeeder
	_rackFeeder : TcaRackFeeder(THIS^);
	RackFeederRef : TcaRackFeederRef;
	
	
	

	
//	// Drive Simple
//	_simpleDrive : TcoDrivesBeckhoff.TcoDriveSimple(THIS^);	
//	SimpleDriveRef	: TcoDrivesBeckhoff.TcoAxisRef;
//		
//	// Axis
//    _horizontalAxis : TcoDrivesBeckhoff.TcoSingleAxis(THIS^);
//	HorizontalAxisRef : TcoDrivesBeckhoff.TcoAxisRef;
//	
//    _vertikalAxis : TcoDrivesBeckhoff.TcoSingleAxis(THIS^);
//	VertikalAxisRef : TcoDrivesBeckhoff.TcoAxisRef;
//	
//    _telekopAxis : TcoDrivesBeckhoff.TcoSingleAxis(THIS^);
//	TeleskopAxisRef	: TcoDrivesBeckhoff.TcoAxisRef;
//	
//    {attribute addProperty Name "<#Test positions#>"}
//    _positions : Handling_Positions(THIS^);
//	
//	
//	// Digital Inouts
//	_digitalInput		: TcoDi(THIS^);
//	
//	
//	_enable1			: BOOL := TRUE;
//	_enablePositive1    : BOOL := TRUE;
//	_enableNegative1    : BOOL := TRUE;
//	_calibrationCam1    : BOOL := TRUE;
//	
//	
//	_position			: LREAL :=1400;
//	_velocity			: LREAL :=1400;
//	_deceleration		: LREAL :=5000;
//	_acceleration		: LREAL :=5000;
//	_jerk				: LREAL :=15000;
	

END_VAR

// TwinSAFE
_TwinSAFE(ref := TwinSAFERef);
_TwinSAFE.Service();

// SafteyGate
_safetyGate_A(ref := SafetyGateRef_A);
_safetyGate_A.Service();
_safetyGate_B(ref := SafetyGateRef_B);
_safetyGate_B.Service();

//RackFeeder
_rackFeeder(ref := RackFeederRef);
_rackFeeder.Service();

// SegementDoor
_segmentDoor_A(ref := SegmentDoorRef_A);
_segmentDoor_A.Service();

_segmentDoor_B(ref := SegmentDoorRef_B);
_segmentDoor_B.Service();


//_segmentDoor(ref := SegmentDoorRef);
//_segmentDoor.Service();



// axis
//_simpleDrive(inEnable := _enable1,
//    inEnablePositive := _enablePositive1,
//    inEnableNegative := _enableNegative1,
//    inCalibrationCam := _calibrationCam1,
//    inoAxisRef := SimpleDriveRef);
//_simpleDrive.Service();
//
//
//_horizontalAxis(inEnable := _enable1,
//    inEnablePositive := _enablePositive1,
//    inEnableNegative := _enableNegative1,
//    inCalibrationCam := _calibrationCam1,
//    refAxis := HorizontalAxisRef,
//	inoPositions:= _positions);	
//_horizontalAxis.Service();	


// sensor
//_sensorLeft(ref := SensorLeftRef);
//_sensorLeft.Service();
//
//_sensorRight(ref := SensorRightRef);
//_sensorRight.Service();

PROPERTY HorizontalAxis :  REFERENCE TO TcoSingleAxis
GET
//HorizontalAxis REF= _horizontalAxis;
END_GET
END_PROPERTY

END_FUNCTION_BLOCK

// ---- Program/MAIN.TcPOU
PROGRAM MAIN
VAR
	_Peripherie	: Peripherie;
END_VAR

_Peripherie.Run();
_Peripherie.RtcSynchronize(TRUE, '', 60);

END_PROGRAM

// ---- Program/Handling/Sequences/Handling_TeachRack.TcPOU
FUNCTION_BLOCK Handling_TeachRack EXTENDS TcoCore.TcoSequencer
VAR	
	_o : TcoCore.TcoSequencerObserver(THIS^);	
	
	_dialog : TcoCore.TcoDialog(THIS^);
	_dialogWithInput        : TcoCore.TcoInputDialog(THIS^);
	
    _customizedContentInput	: Handling_TeachRack_DlgContent(THIS^);

END_VAR

PROPERTY Components : REFERENCE TO Handling_Components
GET
VAR
    _parent : POINTER TO Handling;
END_VAR
IF __QUERYPOINTER(_ParentObject,_parent) THEN // Check if _Parent is Station001
	Components REF= _parent^._components;              // If the check is successful dereference a pointer. simlar to THIS^ or SUPER^
END_IF
END_GET
END_PROPERTY

(*~
	<docu>
		<summary>
			Main method of the sequener. Custom code needs to be placed here. The sequencer is executed by call of InstanceName.Run() method.
			This method is abstract, and it must be overridden in derived block.
		</summary>
	</docu>
~*)
METHOD PROTECTED  Main : BOOL
VAR	
	ErrorStep				: INT := 1000; 
	FinishStep				: INT := 1000;	
END_VAR
THIS^.Observer := _o;

IF (Step(0, TRUE, 'STEP 0')) THEN
	
	_dialogWithInput.Show(refContent:=_customizedContentInput)
         .WithType(eDialogType.Question)
         .WithOk()
         .WithCaption('Set Data for teaching Rack')
         .WithText('Check or Change Values for teaching the Rack');
   
	IF(_dialogWithInput.Answer = TcoCore.eInputDialogAnswer.OK) THEN RequestStep(100); _dialog.Restore(); END_IF;
    IF(_dialogWithInput.Answer = TcoCore.eInputDialogAnswer.No) THEN RequestStep(3000); _dialog.Restore(); END_IF;

END_IF;







